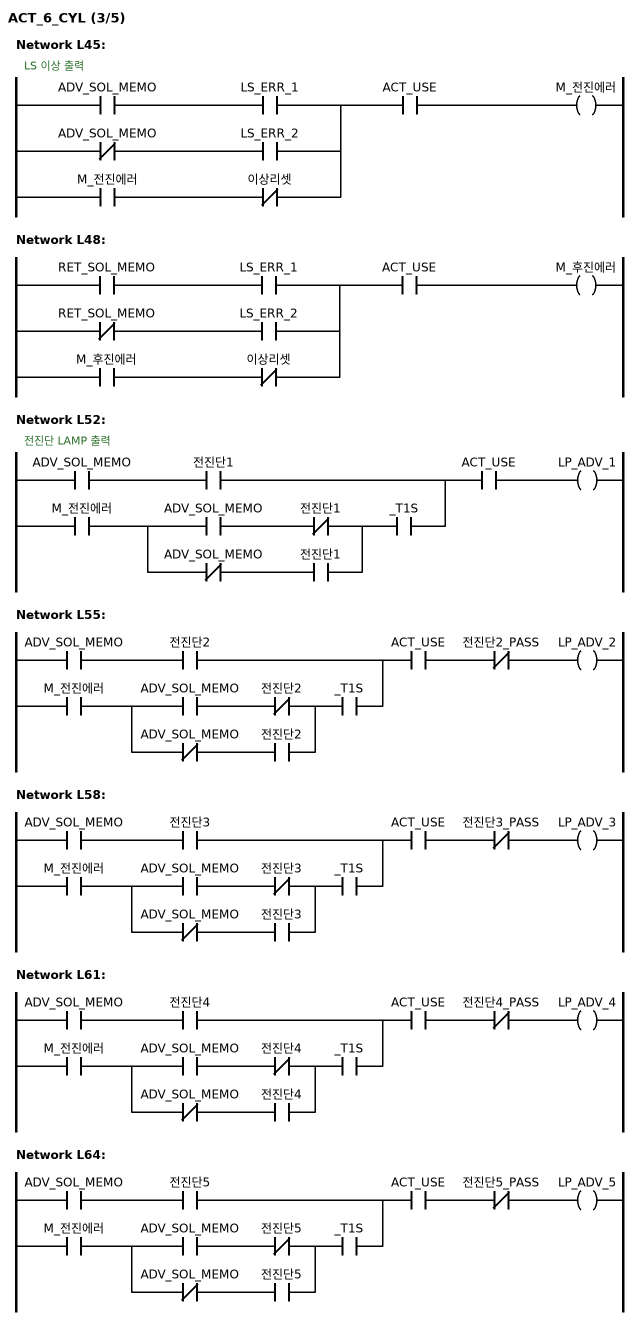
(* [picture p24: ACT_6_CYL rungs L45-L64] *)
(* LS 이상 출력 *)
(* Rung L45 *)
M_전진에러 := ((ADV_SOL_MEMO AND LS_ERR_1) OR (NOT ADV_SOL_MEMO AND LS_ERR_2) OR (M_전진에러 AND NOT 이상리셋)) AND ACT_USE;
(* Rung L48 *)
M_후진에러 := ((RET_SOL_MEMO AND LS_ERR_1) OR (NOT RET_SOL_MEMO AND LS_ERR_2) OR (M_후진에러 AND NOT 이상리셋)) AND ACT_USE;
(* 전진단 LAMP 출력 *)
(* Rung L52 *)
LP_ADV_1 := ((ADV_SOL_MEMO AND 전진단1) OR (M_전진에러 AND ((ADV_SOL_MEMO AND NOT 전진단1) OR (NOT ADV_SOL_MEMO AND 전진단1)) AND _T1S)) AND ACT_USE;
(* Rung L55 *)
LP_ADV_2 := ((ADV_SOL_MEMO AND 전진단2) OR (M_전진에러 AND ((ADV_SOL_MEMO AND NOT 전진단2) OR (NOT ADV_SOL_MEMO AND 전진단2)) AND _T1S)) AND ACT_USE AND NOT 전진단2_PASS;
(* Rung L58 *)
LP_ADV_3 := ((ADV_SOL_MEMO AND 전진단3) OR (M_전진에러 AND ((ADV_SOL_MEMO AND NOT 전진단3) OR (NOT ADV_SOL_MEMO AND 전진단3)) AND _T1S)) AND ACT_USE AND NOT 전진단3_PASS;
(* Rung L61 *)
LP_ADV_4 := ((ADV_SOL_MEMO AND 전진단4) OR (M_전진에러 AND ((ADV_SOL_MEMO AND NOT 전진단4) OR (NOT ADV_SOL_MEMO AND 전진단4)) AND _T1S)) AND ACT_USE AND NOT 전진단4_PASS;
(* Rung L64 *)
LP_ADV_5 := ((ADV_SOL_MEMO AND 전진단5) OR (M_전진에러 AND ((ADV_SOL_MEMO AND NOT 전진단5) OR (NOT ADV_SOL_MEMO AND 전진단5)) AND _T1S)) AND ACT_USE AND NOT 전진단5_PASS;

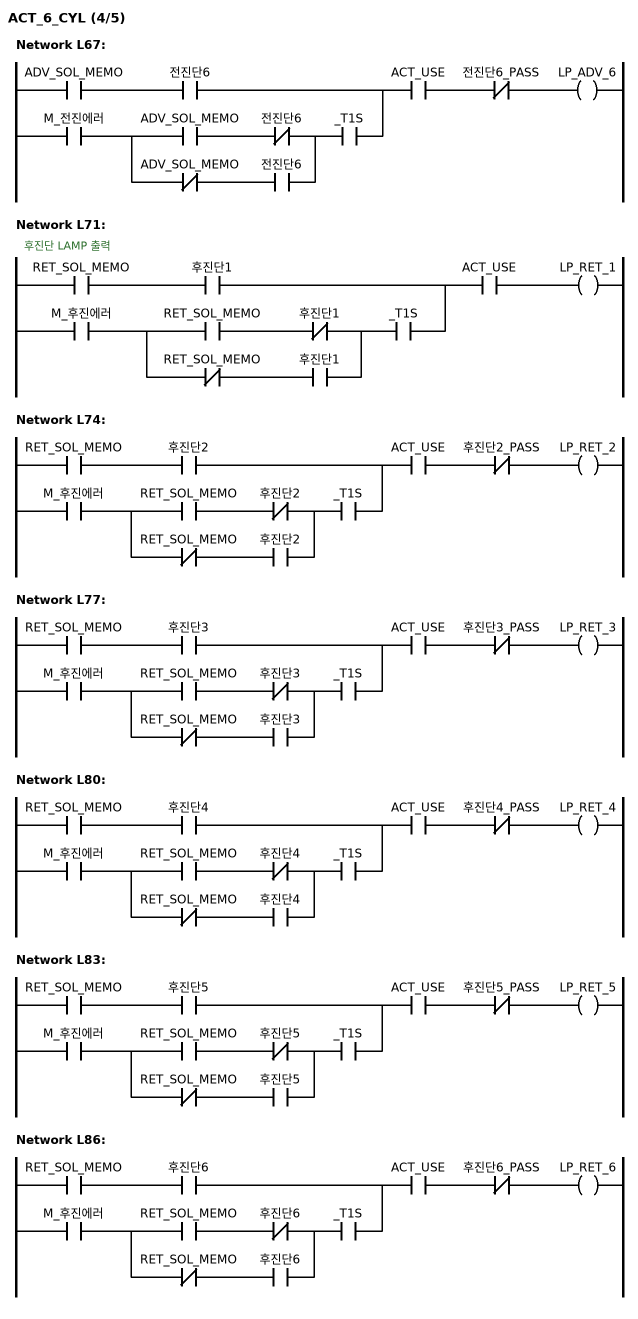
(* Rung L67 *)
LP_ADV_6 := ((ADV_SOL_MEMO AND 전진단6) OR (M_전진에러 AND ((ADV_SOL_MEMO AND NOT 전진단6) OR (NOT ADV_SOL_MEMO AND 전진단6)) AND _T1S)) AND ACT_USE AND NOT 전진단6_PASS;
(* 후진단 LAMP 출력 *)
(* Rung L71 *)
LP_RET_1 := ((RET_SOL_MEMO AND 후진단1) OR (M_후진에러 AND ((RET_SOL_MEMO AND NOT 후진단1) OR (NOT RET_SOL_MEMO AND 후진단1)) AND _T1S)) AND ACT_USE;
(* Rung L74 *)
LP_RET_2 := ((RET_SOL_MEMO AND 후진단2) OR (M_후진에러 AND ((RET_SOL_MEMO AND NOT 후진단2) OR (NOT RET_SOL_MEMO AND 후진단2)) AND _T1S)) AND ACT_USE AND NOT 후진단2_PASS;
(* Rung L77 *)
LP_RET_3 := ((RET_SOL_MEMO AND 후진단3) OR (M_후진에러 AND ((RET_SOL_MEMO AND NOT 후진단3) OR (NOT RET_SOL_MEMO AND 후진단3)) AND _T1S)) AND ACT_USE AND NOT 후진단3_PASS;
(* Rung L80 *)
LP_RET_4 := ((RET_SOL_MEMO AND 후진단4) OR (M_후진에러 AND ((RET_SOL_MEMO AND NOT 후진단4) OR (NOT RET_SOL_MEMO AND 후진단4)) AND _T1S)) AND ACT_USE AND NOT 후진단4_PASS;
(* Rung L83 *)
LP_RET_5 := ((RET_SOL_MEMO AND 후진단5) OR (M_후진에러 AND ((RET_SOL_MEMO AND NOT 후진단5) OR (NOT RET_SOL_MEMO AND 후진단5)) AND _T1S)) AND ACT_USE AND NOT 후진단5_PASS;
(* Rung L86 *)
LP_RET_6 := ((RET_SOL_MEMO AND 후진단6) OR (M_후진에러 AND ((RET_SOL_MEMO AND NOT 후진단6) OR (NOT RET_SOL_MEMO AND 후진단6)) AND _T1S)) AND ACT_USE AND NOT 후진단6_PASS;

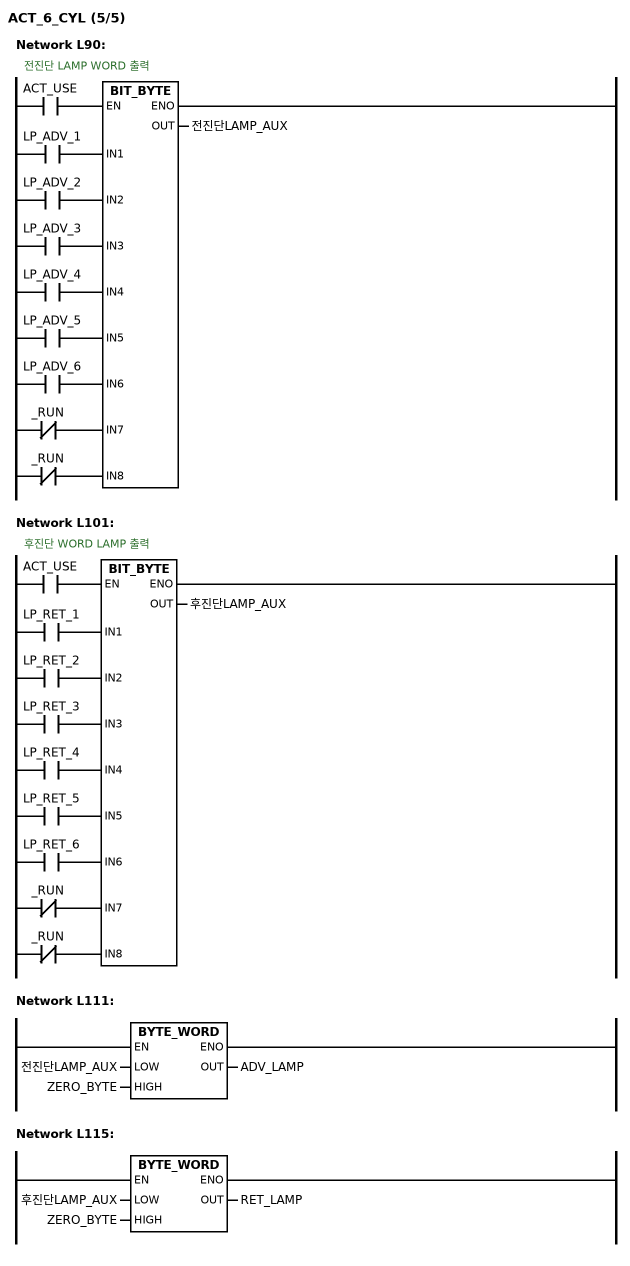
(* 전진단 LAMP WORD 출력 *)
(* Rung L90 *)
IF ACT_USE THEN
    전진단LAMP_AUX := BIT_BYTE(LP_ADV_1, LP_ADV_2, LP_ADV_3, LP_ADV_4, LP_ADV_5, LP_ADV_6, NOT _RUN, NOT _RUN);
END_IF;
(* 후진단 WORD LAMP 출력 *)
(* Rung L101 *)
IF ACT_USE THEN
    후진단LAMP_AUX := BIT_BYTE(LP_RET_1, LP_RET_2, LP_RET_3, LP_RET_4, LP_RET_5, LP_RET_6, NOT _RUN, NOT _RUN);
END_IF;
(* Rung L111 *)
ADV_LAMP := BYTE_WORD(LOW := 전진단LAMP_AUX, HIGH := ZERO_BYTE);
(* Rung L115 *)
RET_LAMP := BYTE_WORD(LOW := 후진단LAMP_AUX, HIGH := ZERO_BYTE);
END_FUNCTION_BLOCK

FUNCTION_BLOCK ACT_10_CYL
VAR_INPUT
    사용유무 : BOOL;
    운전준비 : BOOL;
    전진보조 : BOOL;
    후진보조 : BOOL;
    전진단수량 : UINT;
    후진단수량 : UINT;
    전진단1 : BOOL;
    후진단1 : BOOL;
    전진단2 : BOOL;
    후진단2 : BOOL;
    전진단3 : BOOL;
    후진단3 : BOOL;
    전진단4 : BOOL;
    후진단4 : BOOL;
    전진단5 : BOOL;
    후진단5 : BOOL;
    전진단6 : BOOL;
    후진단6 : BOOL;
    전진단7 : BOOL;
    후진단7 : BOOL;
    전진단8 : BOOL;
    후진단8 : BOOL;
    전진단9 : BOOL;
    후진단9 : BOOL;
    전진단10 : BOOL;
    후진단10 : BOOL;
    전진단_지연시간 : TIME;
    후진단_지연시간 : TIME;
    LS_ERR1_지연시간 : TIME;
    LS_ERR2_지연시간 : TIME;
    이상리셋 : BOOL;
END_VAR
VAR_OUTPUT
    SOL_ADV_출력 : BOOL;
    SOL_RET_출력 : BOOL;
    M_전진단 : BOOL;
    M_후진단 : BOOL;
    M_전진에러 : BOOL;
    M_후진에러 : BOOL;
    ADV_LAMP : WORD;
    RET_LAMP : WORD;
END_VAR
VAR
    ACT_USE : BOOL;
    ADV_END_TIME : TON;
    ADV_SOL_MEMO : BOOL;
    ERR_TIME1 : TON;
    LP_ADV_1 : BOOL;
    LP_ADV_10 : BOOL;
    LP_ADV_2 : BOOL;
    LP_ADV_3 : BOOL;
    LP_ADV_4 : BOOL;
    LP_ADV_5 : BOOL;
    LP_ADV_6 : BOOL;
    LP_ADV_7 : BOOL;
    LP_ADV_8 : BOOL;
    LP_ADV_9 : BOOL;
    LP_RET_1 : BOOL;
    LP_RET_10 : BOOL;
    LP_RET_2 : BOOL;
    LP_RET_3 : BOOL;
    LP_RET_4 : BOOL;
    LP_RET_5 : BOOL;
    LP_RET_6 : BOOL;
    LP_RET_7 : BOOL;
    LP_RET_8 : BOOL;
    LP_RET_9 : BOOL;
    LS_ERR_1 : BOOL;
    LS_ERR_2 : BOOL;
    RET_END_TIME : TON;
    RET_END_TIME1 : TON;
    RET_END_TIME2 : TON;
    RET_ERR_TIME : TON;
    RET_SOL_MEMO : BOOL;
    전진단10_PASS : BOOL;
    전진단2_PASS : BOOL;
    전진단3_PASS : BOOL;
    전진단4_PASS : BOOL;
    전진단5_PASS : BOOL;
    전진단6_PASS : BOOL;
    전진단7_PASS : BOOL;
    전진단8_PASS : BOOL;
    전진단9_PASS : BOOL;
    전진단LAMP_H_AUX : BYTE;
    전진단LAMP_L_AUX : BYTE;
    후진단10_PASS : BOOL;
    후진단2_PASS : BOOL;
    후진단3_PASS : BOOL;
    후진단4_PASS : BOOL;
    후진단5_PASS : BOOL;
    후진단6_PASS : BOOL;
    후진단7_PASS : BOOL;
    후진단8_PASS : BOOL;
    후진단9_PASS : BOOL;
    후진단LAMP_H_AUX : BYTE;
    후진단LAMP_L_AUX : BYTE;
END_VAR

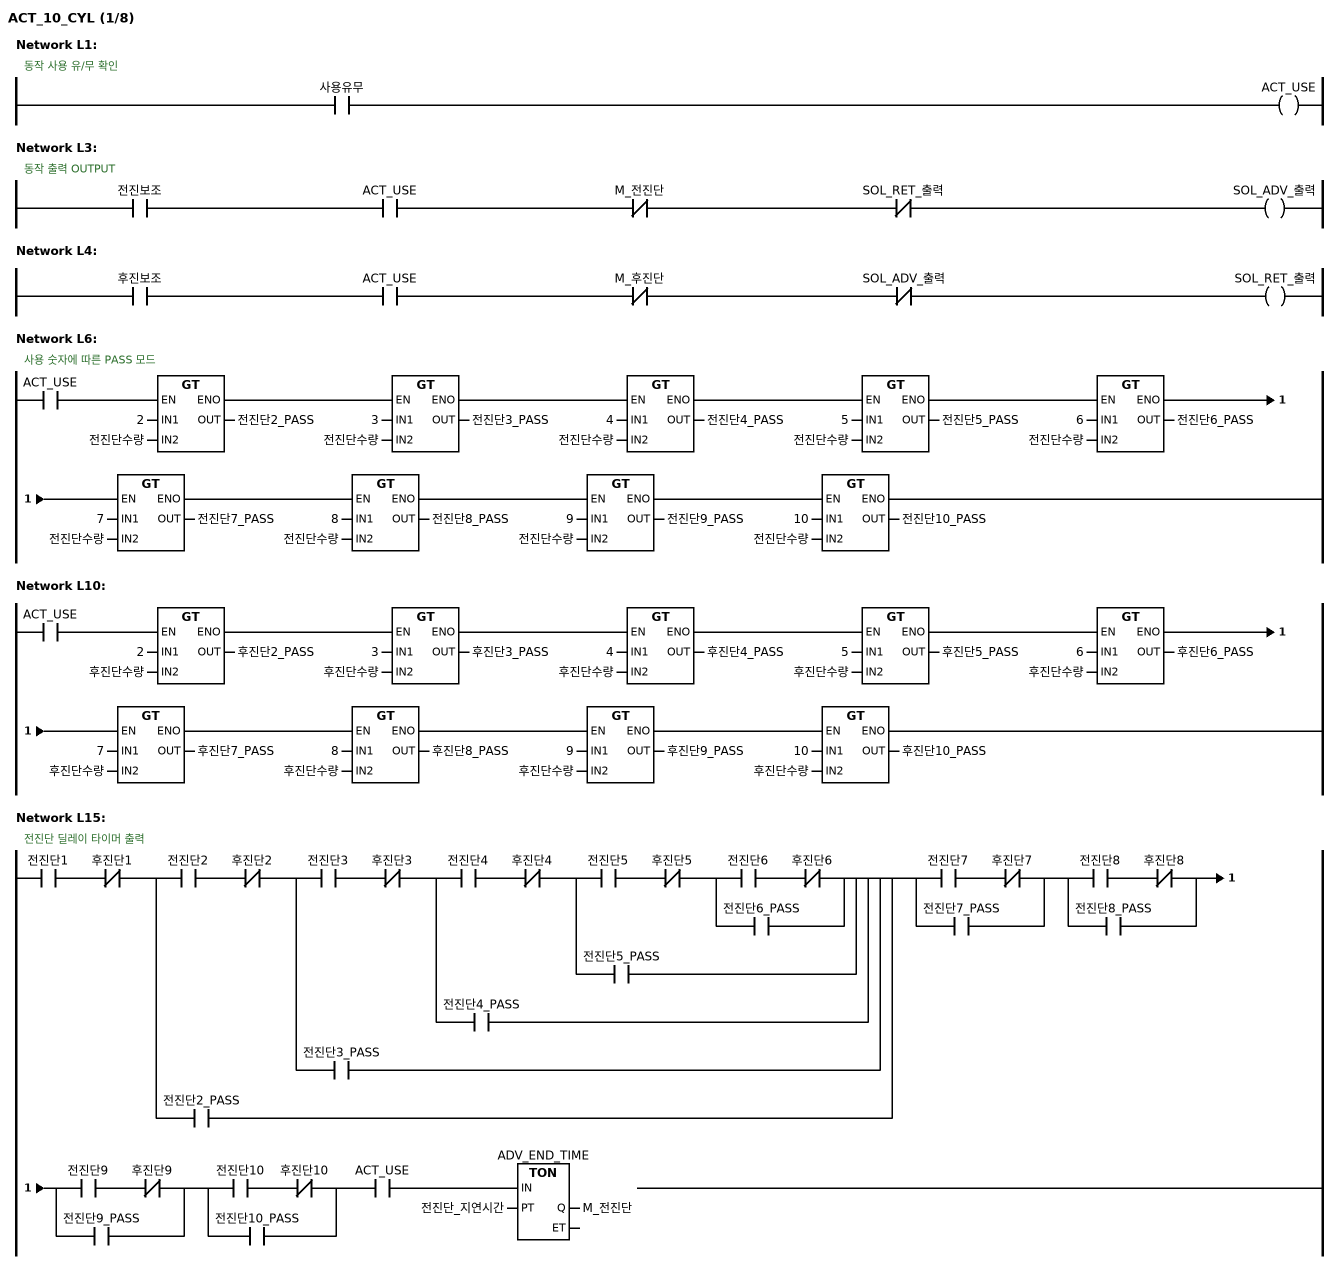
(* 동작 사용 유/무 확인 *)
(* Rung L1 *)
ACT_USE := 사용유무;
(* 동작 출력 OUTPUT *)
(* Rung L3 *)
SOL_ADV_출력 := 전진보조 AND ACT_USE AND NOT M_전진단 AND NOT SOL_RET_출력;
(* Rung L4 *)
SOL_RET_출력 := 후진보조 AND ACT_USE AND NOT M_후진단 AND NOT SOL_ADV_출력;
(* 사용 숫자에 따른 PASS 모드 *)
(* Rung L6 *)
IF ACT_USE THEN
    전진단2_PASS := 2 > 전진단수량;
    전진단3_PASS := 3 > 전진단수량;
    전진단4_PASS := 4 > 전진단수량;
    전진단5_PASS := 5 > 전진단수량;
    전진단6_PASS := 6 > 전진단수량;
    전진단7_PASS := 7 > 전진단수량;
    전진단8_PASS := 8 > 전진단수량;
    전진단9_PASS := 9 > 전진단수량;
    전진단10_PASS := 10 > 전진단수량;
END_IF;
(* Rung L10 *)
IF ACT_USE THEN
    후진단2_PASS := 2 > 후진단수량;
    후진단3_PASS := 3 > 후진단수량;
    후진단4_PASS := 4 > 후진단수량;
    후진단5_PASS := 5 > 후진단수량;
    후진단6_PASS := 6 > 후진단수량;
    후진단7_PASS := 7 > 후진단수량;
    후진단8_PASS := 8 > 후진단수량;
    후진단9_PASS := 9 > 후진단수량;
    후진단10_PASS := 10 > 후진단수량;
END_IF;
(* 전진단 딜레이 타이머 출력 *)
(* Rung L15 *)
ADV_END_TIME(IN := 전진단1 AND NOT 후진단1 AND ((전진단2 AND NOT 후진단2 AND ((전진단3 AND NOT 후진단3 AND ((전진단4 AND NOT 후진단4 AND ((전진단5 AND NOT 후진단5 AND ((전진단6 AND NOT 후진단6) OR 전진단6_PASS)) OR 전진단5_PASS)) OR 전진단4_PASS)) OR 전진단3_PASS)) OR 전진단2_PASS) AND ((전진단7 AND NOT 후진단7) OR 전진단7_PASS) AND ((전진단8 AND NOT 후진단8) OR 전진단8_PASS) AND ((전진단9 AND NOT 후진단9) OR 전진단9_PASS) AND ((전진단10 AND NOT 후진단10) OR 전진단10_PASS) AND ACT_USE, PT := 전진단_지연시간, Q => M_전진단);

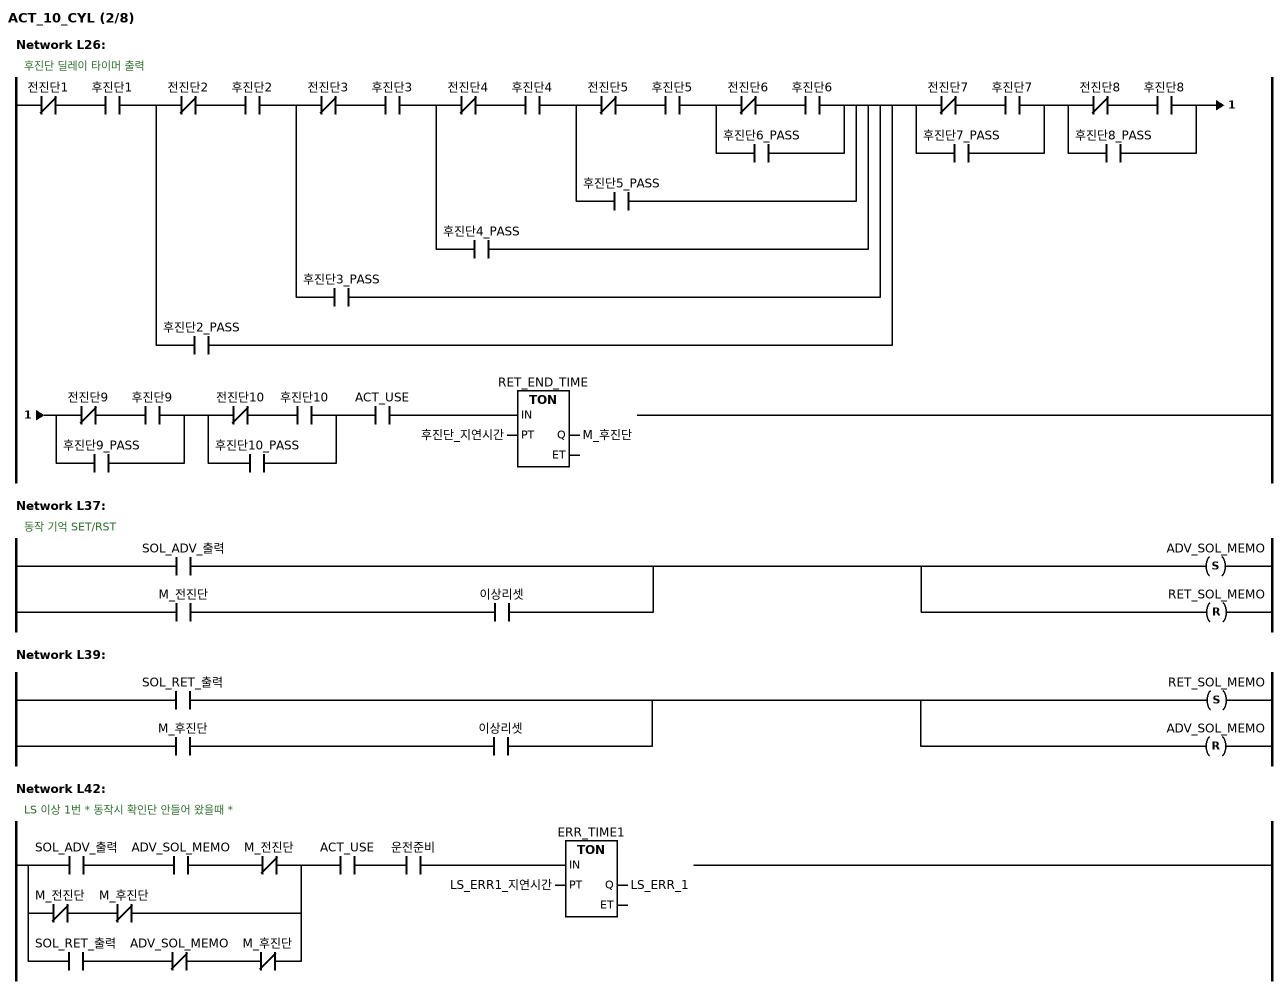
(* 후진단 딜레이 타이머 출력 *)
(* Rung L26 *)
RET_END_TIME(IN := NOT 전진단1 AND 후진단1 AND ((NOT 전진단2 AND 후진단2 AND ((NOT 전진단3 AND 후진단3 AND ((NOT 전진단4 AND 후진단4 AND ((NOT 전진단5 AND 후진단5 AND ((NOT 전진단6 AND 후진단6) OR 후진단6_PASS)) OR 후진단5_PASS)) OR 후진단4_PASS)) OR 후진단3_PASS)) OR 후진단2_PASS) AND ((NOT 전진단7 AND 후진단7) OR 후진단7_PASS) AND ((NOT 전진단8 AND 후진단8) OR 후진단8_PASS) AND ((NOT 전진단9 AND 후진단9) OR 후진단9_PASS) AND ((NOT 전진단10 AND 후진단10) OR 후진단10_PASS) AND ACT_USE, PT := 후진단_지연시간, Q => M_후진단);
(* 동작 기억 SET/RST *)
(* Rung L37 *)
IF SOL_ADV_출력 OR (M_전진단 AND 이상리셋) THEN
    ADV_SOL_MEMO := TRUE;
    RET_SOL_MEMO := FALSE;
END_IF;
(* Rung L39 *)
IF SOL_RET_출력 OR (M_후진단 AND 이상리셋) THEN
    RET_SOL_MEMO := TRUE;
    ADV_SOL_MEMO := FALSE;
END_IF;
(* LS 이상 1번 * 동작시 확인단 안들어 왔을때 * *)
(* Rung L42 *)
ERR_TIME1(IN := ((SOL_ADV_출력 AND ADV_SOL_MEMO AND NOT M_전진단) OR (NOT M_전진단 AND NOT M_후진단) OR (SOL_RET_출력 AND NOT ADV_SOL_MEMO AND NOT M_후진단)) AND ACT_USE AND 운전준비, PT := LS_ERR1_지연시간, Q => LS_ERR_1);

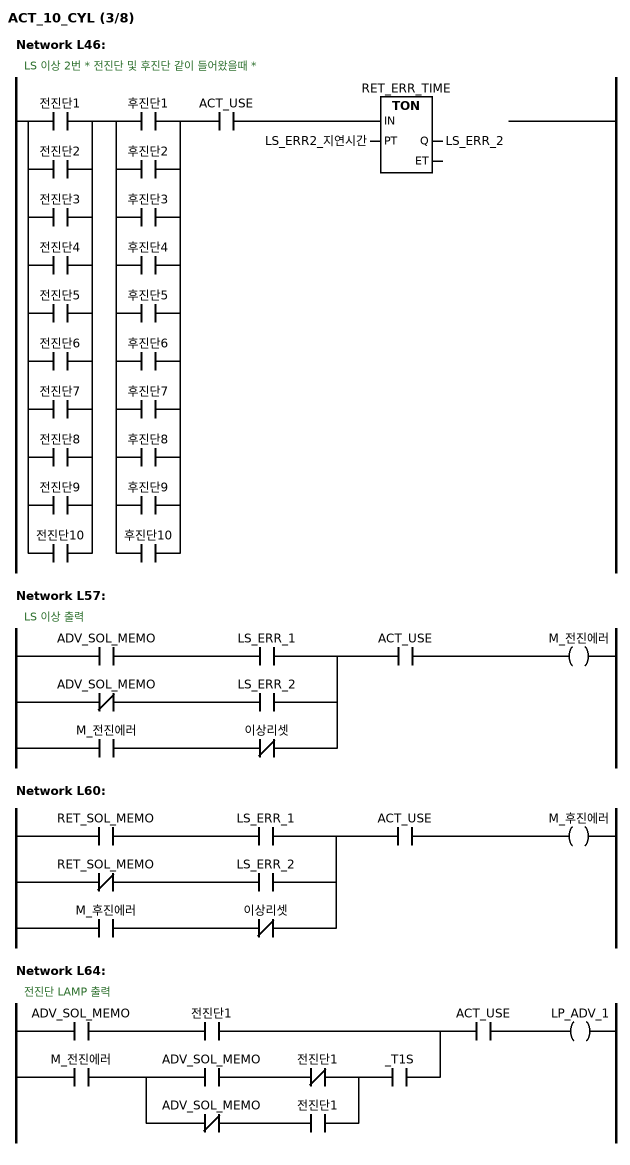
(* LS 이상 2번 * 전진단 및 후진단 같이 들어왔을때 * *)
(* Rung L46 *)
RET_ERR_TIME(IN := (전진단1 OR 전진단2 OR 전진단3 OR 전진단4 OR 전진단5 OR 전진단6 OR 전진단7 OR 전진단8 OR 전진단9 OR 전진단10) AND (후진단1 OR 후진단2 OR 후진단3 OR 후진단4 OR 후진단5 OR 후진단6 OR 후진단7 OR 후진단8 OR 후진단9 OR 후진단10) AND ACT_USE, PT := LS_ERR2_지연시간, Q => LS_ERR_2);
(* LS 이상 출력 *)
(* Rung L57 *)
M_전진에러 := ((ADV_SOL_MEMO AND LS_ERR_1) OR (NOT ADV_SOL_MEMO AND LS_ERR_2) OR (M_전진에러 AND NOT 이상리셋)) AND ACT_USE;
(* Rung L60 *)
M_후진에러 := ((RET_SOL_MEMO AND LS_ERR_1) OR (NOT RET_SOL_MEMO AND LS_ERR_2) OR (M_후진에러 AND NOT 이상리셋)) AND ACT_USE;
(* 전진단 LAMP 출력 *)
(* Rung L64 *)
LP_ADV_1 := ((ADV_SOL_MEMO AND 전진단1) OR (M_전진에러 AND ((ADV_SOL_MEMO AND NOT 전진단1) OR (NOT ADV_SOL_MEMO AND 전진단1)) AND _T1S)) AND ACT_USE;

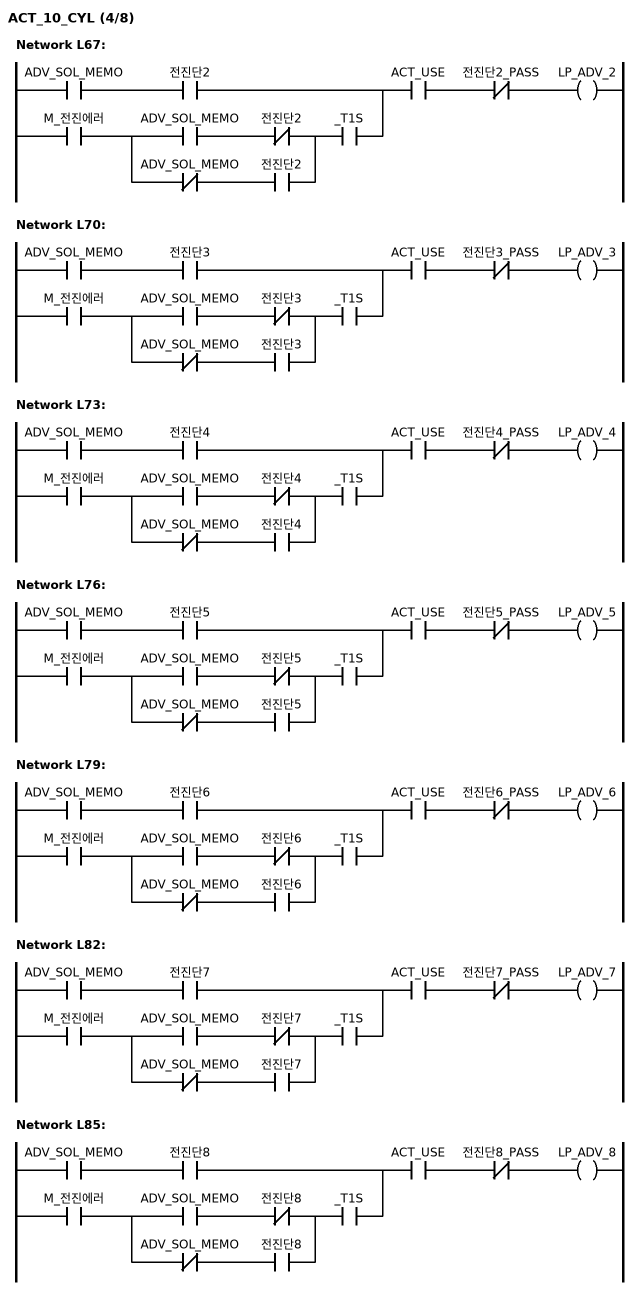
(* Rung L67 *)
LP_ADV_2 := ((ADV_SOL_MEMO AND 전진단2) OR (M_전진에러 AND ((ADV_SOL_MEMO AND NOT 전진단2) OR (NOT ADV_SOL_MEMO AND 전진단2)) AND _T1S)) AND ACT_USE AND NOT 전진단2_PASS;
(* Rung L70 *)
LP_ADV_3 := ((ADV_SOL_MEMO AND 전진단3) OR (M_전진에러 AND ((ADV_SOL_MEMO AND NOT 전진단3) OR (NOT ADV_SOL_MEMO AND 전진단3)) AND _T1S)) AND ACT_USE AND NOT 전진단3_PASS;
(* Rung L73 *)
LP_ADV_4 := ((ADV_SOL_MEMO AND 전진단4) OR (M_전진에러 AND ((ADV_SOL_MEMO AND NOT 전진단4) OR (NOT ADV_SOL_MEMO AND 전진단4)) AND _T1S)) AND ACT_USE AND NOT 전진단4_PASS;
(* Rung L76 *)
LP_ADV_5 := ((ADV_SOL_MEMO AND 전진단5) OR (M_전진에러 AND ((ADV_SOL_MEMO AND NOT 전진단5) OR (NOT ADV_SOL_MEMO AND 전진단5)) AND _T1S)) AND ACT_USE AND NOT 전진단5_PASS;
(* Rung L79 *)
LP_ADV_6 := ((ADV_SOL_MEMO AND 전진단6) OR (M_전진에러 AND ((ADV_SOL_MEMO AND NOT 전진단6) OR (NOT ADV_SOL_MEMO AND 전진단6)) AND _T1S)) AND ACT_USE AND NOT 전진단6_PASS;
(* Rung L82 *)
LP_ADV_7 := ((ADV_SOL_MEMO AND 전진단7) OR (M_전진에러 AND ((ADV_SOL_MEMO AND NOT 전진단7) OR (NOT ADV_SOL_MEMO AND 전진단7)) AND _T1S)) AND ACT_USE AND NOT 전진단7_PASS;
(* Rung L85 *)
LP_ADV_8 := ((ADV_SOL_MEMO AND 전진단8) OR (M_전진에러 AND ((ADV_SOL_MEMO AND NOT 전진단8) OR (NOT ADV_SOL_MEMO AND 전진단8)) AND _T1S)) AND ACT_USE AND NOT 전진단8_PASS;

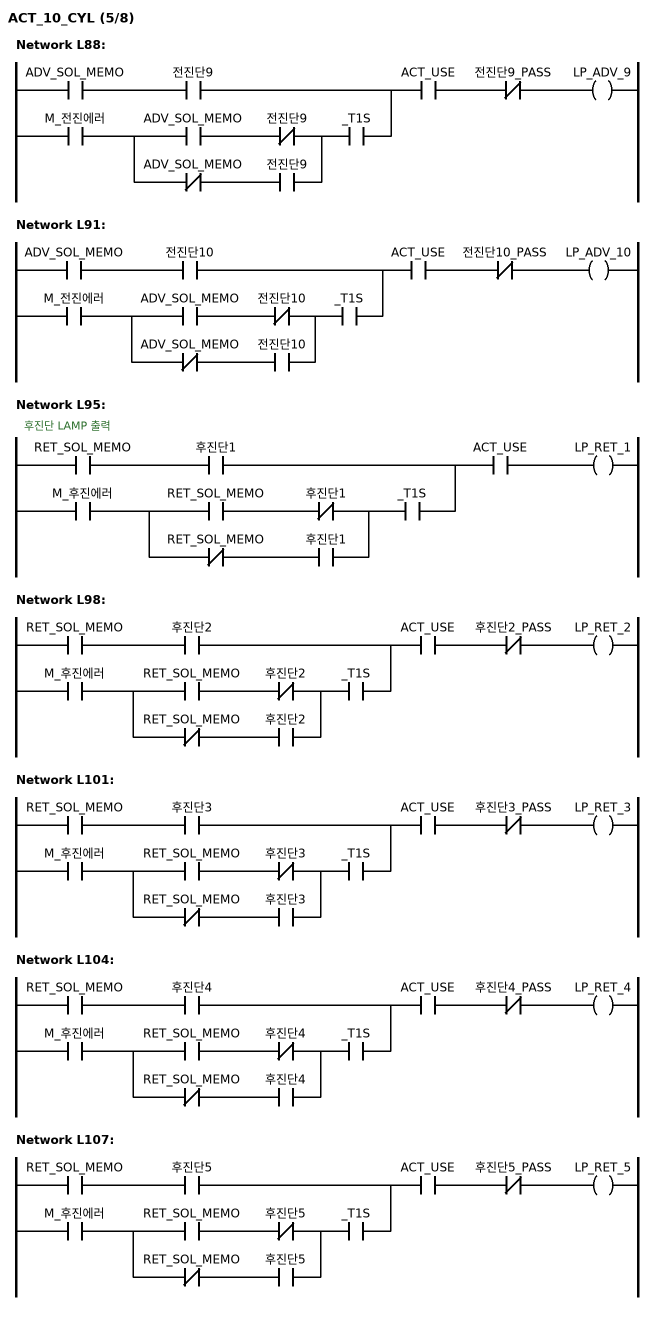
(* Rung L88 *)
LP_ADV_9 := ((ADV_SOL_MEMO AND 전진단9) OR (M_전진에러 AND ((ADV_SOL_MEMO AND NOT 전진단9) OR (NOT ADV_SOL_MEMO AND 전진단9)) AND _T1S)) AND ACT_USE AND NOT 전진단9_PASS;
(* Rung L91 *)
LP_ADV_10 := ((ADV_SOL_MEMO AND 전진단10) OR (M_전진에러 AND ((ADV_SOL_MEMO AND NOT 전진단10) OR (NOT ADV_SOL_MEMO AND 전진단10)) AND _T1S)) AND ACT_USE AND NOT 전진단10_PASS;
(* 후진단 LAMP 출력 *)
(* Rung L95 *)
LP_RET_1 := ((RET_SOL_MEMO AND 후진단1) OR (M_후진에러 AND ((RET_SOL_MEMO AND NOT 후진단1) OR (NOT RET_SOL_MEMO AND 후진단1)) AND _T1S)) AND ACT_USE;
(* Rung L98 *)
LP_RET_2 := ((RET_SOL_MEMO AND 후진단2) OR (M_후진에러 AND ((RET_SOL_MEMO AND NOT 후진단2) OR (NOT RET_SOL_MEMO AND 후진단2)) AND _T1S)) AND ACT_USE AND NOT 후진단2_PASS;
(* Rung L101 *)
LP_RET_3 := ((RET_SOL_MEMO AND 후진단3) OR (M_후진에러 AND ((RET_SOL_MEMO AND NOT 후진단3) OR (NOT RET_SOL_MEMO AND 후진단3)) AND _T1S)) AND ACT_USE AND NOT 후진단3_PASS;
(* Rung L104 *)
LP_RET_4 := ((RET_SOL_MEMO AND 후진단4) OR (M_후진에러 AND ((RET_SOL_MEMO AND NOT 후진단4) OR (NOT RET_SOL_MEMO AND 후진단4)) AND _T1S)) AND ACT_USE AND NOT 후진단4_PASS;
(* Rung L107 *)
LP_RET_5 := ((RET_SOL_MEMO AND 후진단5) OR (M_후진에러 AND ((RET_SOL_MEMO AND NOT 후진단5) OR (NOT RET_SOL_MEMO AND 후진단5)) AND _T1S)) AND ACT_USE AND NOT 후진단5_PASS;

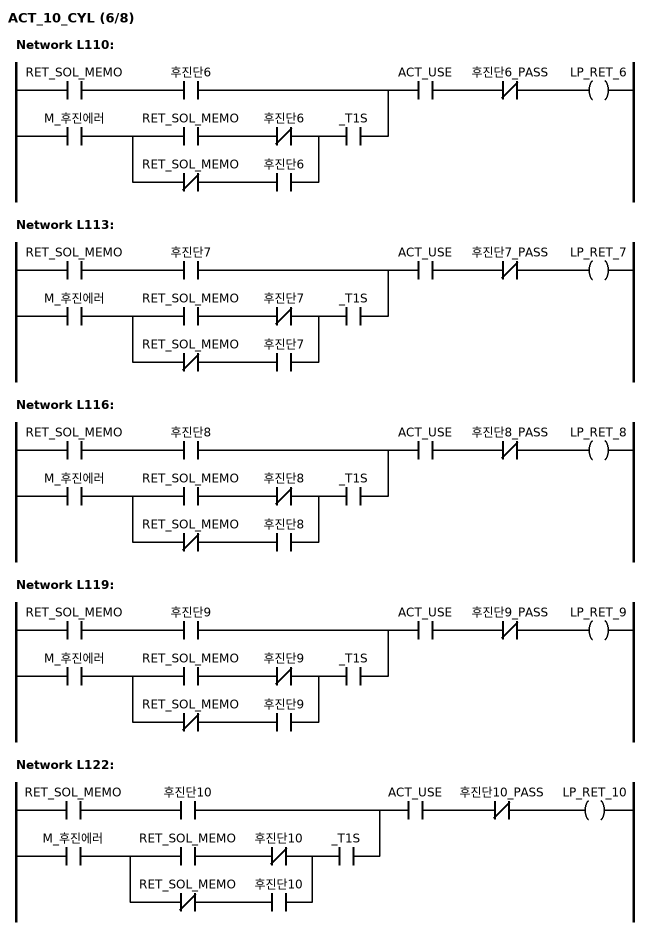
(* Rung L110 *)
LP_RET_6 := ((RET_SOL_MEMO AND 후진단6) OR (M_후진에러 AND ((RET_SOL_MEMO AND NOT 후진단6) OR (NOT RET_SOL_MEMO AND 후진단6)) AND _T1S)) AND ACT_USE AND NOT 후진단6_PASS;
(* Rung L113 *)
LP_RET_7 := ((RET_SOL_MEMO AND 후진단7) OR (M_후진에러 AND ((RET_SOL_MEMO AND NOT 후진단7) OR (NOT RET_SOL_MEMO AND 후진단7)) AND _T1S)) AND ACT_USE AND NOT 후진단7_PASS;
(* Rung L116 *)
LP_RET_8 := ((RET_SOL_MEMO AND 후진단8) OR (M_후진에러 AND ((RET_SOL_MEMO AND NOT 후진단8) OR (NOT RET_SOL_MEMO AND 후진단8)) AND _T1S)) AND ACT_USE AND NOT 후진단8_PASS;
(* Rung L119 *)
LP_RET_9 := ((RET_SOL_MEMO AND 후진단9) OR (M_후진에러 AND ((RET_SOL_MEMO AND NOT 후진단9) OR (NOT RET_SOL_MEMO AND 후진단9)) AND _T1S)) AND ACT_USE AND NOT 후진단9_PASS;
(* Rung L122 *)
LP_RET_10 := ((RET_SOL_MEMO AND 후진단10) OR (M_후진에러 AND ((RET_SOL_MEMO AND NOT 후진단10) OR (NOT RET_SOL_MEMO AND 후진단10)) AND _T1S)) AND ACT_USE AND NOT 후진단10_PASS;

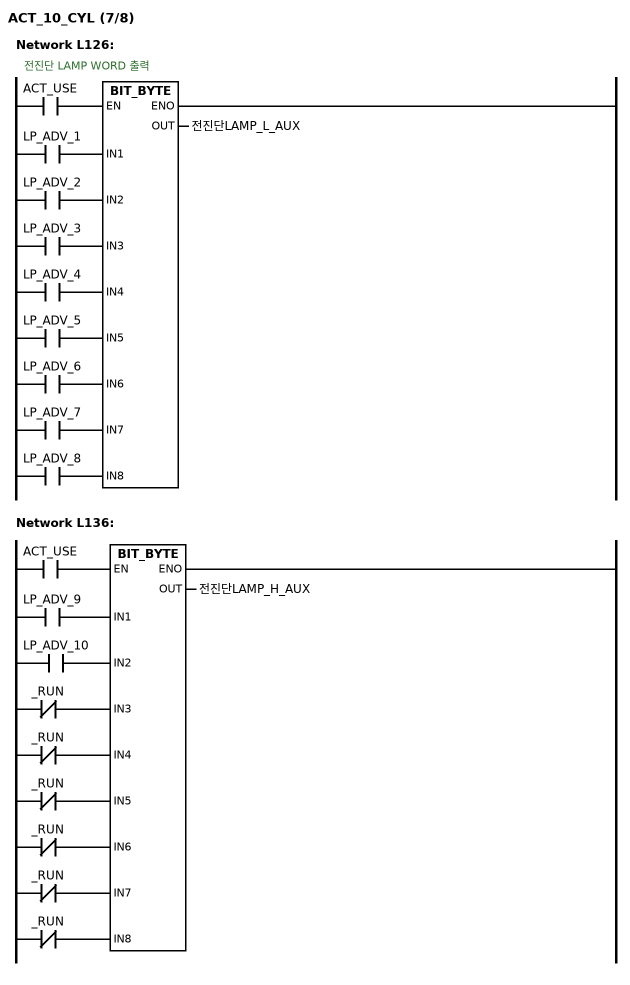
(* 전진단 LAMP WORD 출력 *)
(* Rung L126 *)
IF ACT_USE THEN
    전진단LAMP_L_AUX := BIT_BYTE(LP_ADV_1, LP_ADV_2, LP_ADV_3, LP_ADV_4, LP_ADV_5, LP_ADV_6, LP_ADV_7, LP_ADV_8);
END_IF;
(* Rung L136 *)
IF ACT_USE THEN
    전진단LAMP_H_AUX := BIT_BYTE(LP_ADV_9, LP_ADV_10, NOT _RUN, NOT _RUN, NOT _RUN, NOT _RUN, NOT _RUN, NOT _RUN);
END_IF;

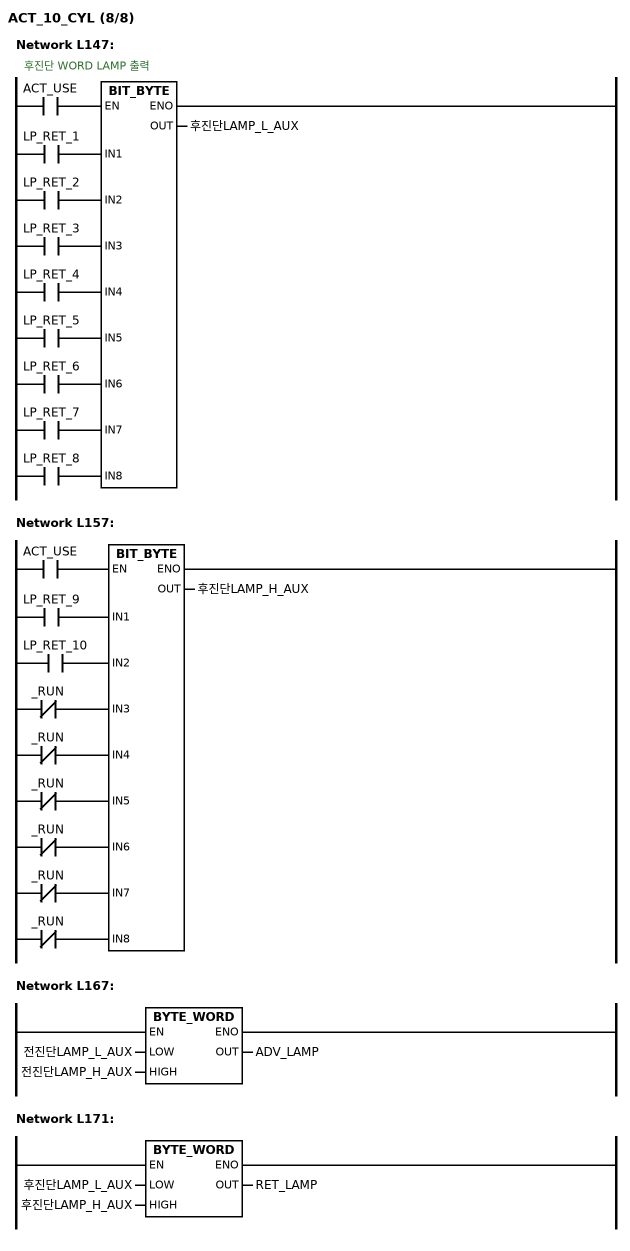
(* 후진단 WORD LAMP 출력 *)
(* Rung L147 *)
IF ACT_USE THEN
    후진단LAMP_L_AUX := BIT_BYTE(LP_RET_1, LP_RET_2, LP_RET_3, LP_RET_4, LP_RET_5, LP_RET_6, LP_RET_7, LP_RET_8);
END_IF;
(* Rung L157 *)
IF ACT_USE THEN
    후진단LAMP_H_AUX := BIT_BYTE(LP_RET_9, LP_RET_10, NOT _RUN, NOT _RUN, NOT _RUN, NOT _RUN, NOT _RUN, NOT _RUN);
END_IF;
(* Rung L167 *)
ADV_LAMP := BYTE_WORD(LOW := 전진단LAMP_L_AUX, HIGH := 전진단LAMP_H_AUX);
(* Rung L171 *)
RET_LAMP := BYTE_WORD(LOW := 후진단LAMP_L_AUX, HIGH := 후진단LAMP_H_AUX);
END_FUNCTION_BLOCK

PROGRAM 운전모드 (* task: 스캔 프로그램 *)
VAR_EXTERNAL
    AWAYS_ON : BOOL; (* AT %MW3.1 *)
    CLOCK_BIT_0_5Sec : BOOL; (* AT %MW0.3 *)
    EGIS_EJS : BOOL;
    GATE10_M_도어_잠김 : BOOL; (* AT %MW409.3 *)
    GATE10_M_비상정지 : BOOL; (* AT %MW409.7 *)
    GATE10_M_이상_리셋 : BOOL; (* AT %MW409.0 *)
    GATE10_M_정상 : BOOL; (* AT %MW409.4 *)
    GATE11_M_이상_리셋 : BOOL; (* AT %MW410.0 *)
    GATE11_M_정상 : BOOL; (* AT %MW410.4 *)
    GATE12_M_이상_리셋 : BOOL; (* AT %MW411.0 *)
    GATE12_M_정상 : BOOL; (* AT %MW411.4 *)
    MCP_EPB_비상정지1 : BOOL; (* AT %MW87635.0 *) (* 입력 접점 00 *)
    MCP_EPB_비상정지2 : BOOL; (* AT %MW87635.1 *) (* 입력 접점 01 *)
    MCP_KSW_MES_OFF : BOOL; (* AT %MW87631.4 *) (* 입력 접점 04 *)
    MCP_KSW_MES_ON : BOOL; (* AT %MW87631.5 *) (* 입력 접점 05 *)
    MCP_MC1_OUTPUT_PWR_ON : BOOL; (* AT %MW97636.0 *) (* 출력 접점 00 *)
    MCP_M_램프_테스트 : BOOL; (* AT %MW350.6 *)
    MCP_M_부저_정지 : BOOL; (* AT %MW350.5 *)
    MCP_M_비상정지 : BOOL; (* AT %MW350.7 *)
    MCP_M_수동_모드 : BOOL; (* AT %MW350.1 *)
    MCP_M_운전준비_ON : BOOL; (* AT %MW350.0 *)
    MCP_M_이상_리셋 : BOOL; (* AT %MW350.4 *)
    MCP_M_자동_START : BOOL; (* AT %MW350.3 *)
    MCP_M_자동_모드 : BOOL; (* AT %MW350.2 *)
    MCP_PBL_101_자동_운전 : BOOL; (* AT %MW87630.4 *) (* 입력 접점 04 *)
    MCP_PBL_101_자동_운전_LP : BOOL; (* AT %MW97633.1 *) (* 출력 접점 01 *)
    MCP_PBL_102_자동_운전 : BOOL; (* AT %MW87630.7 *) (* 입력 접점 07 *)
    MCP_PBL_102_자동_운전_LP : BOOL; (* AT %MW97633.2 *) (* 출력 접점 02 *)
    MCP_PBL_103_4_자동_운전 : BOOL; (* AT %MW87630.10 *) (* 입력 접점 10 *)
    MCP_PBL_103_4_자동_운전_LP : BOOL; (* AT %MW97633.3 *) (* 출력 접점 03 *)
    MCP_PBL_운전준비_ON : BOOL; (* AT %MW87630.0 *) (* 입력 접점 00 *)
    MCP_PBL_운전준비_ON_LP : BOOL; (* AT %MW97633.0 *) (* 출력 접점 00 *)
    MCP_PB_이상_리셋 : BOOL; (* AT %MW87630.1 *) (* 입력 접점 01 *)
    MCP_SPB_램프_테스트 : BOOL; (* AT %MW87631.2 *) (* 입력 접점 02 *)
    MCP_SPB_부저_정지 : BOOL; (* AT %MW87631.3 *) (* 입력 접점 03 *)
    MCP_SPK_MEL1 : BOOL; (* AT %MW97633.8 *) (* 출력 접점 08 *)
    MCP_SSP_101_수동_선택 : BOOL; (* AT %MW87630.2 *) (* 입력 접점 02 *)
    MCP_SSP_101_자동_선택 : BOOL; (* AT %MW87630.3 *) (* 입력 접점 03 *)
    MCP_TL_GREEN_LAMP : BOOL; (* AT %MW97633.6 *) (* 출력 접점 06 *)
    MCP_TL_RED_LAMP : BOOL; (* AT %MW97633.4 *) (* 출력 접점 04 *)
    MCP_TL_YELLOW_LAMP : BOOL; (* AT %MW97633.5 *) (* 출력 접점 05 *)
    MCP_타워_부저 : BOOL; (* AT %MW97633.7 *) (* 출력 접점 07 *)
    S101_M_수동_모드 : BOOL; (* AT %MW1000.3 *)
    S101_M_운전준비_ON : BOOL; (* AT %MW1000.0 *)
    S101_M_자동_START : BOOL; (* AT %MW1000.5 *)
    S101_M_자동_모드 : BOOL; (* AT %MW1000.1 *)
    S101_M_자동_운전중 : BOOL; (* AT %MW1000.4 *)
    S101_M_총괄_비상정지_이상 : BOOL; (* AT %MW1009.1 *)
    S101_M_총괄_이상 : BOOL; (* AT %MW1009.0 *)
    S102_M_수동_모드 : BOOL; (* AT %MW1500.3 *)
    S102_M_운전준비_ON : BOOL; (* AT %MW1500.0 *)
    S102_M_자동_START : BOOL; (* AT %MW1500.5 *)
    S102_M_자동_모드 : BOOL; (* AT %MW1500.1 *)
    S102_M_자동_운전중 : BOOL; (* AT %MW1500.4 *)
    S102_M_총괄_비상정지_이상 : BOOL; (* AT %MW1509.1 *)
    S102_M_총괄_이상 : BOOL; (* AT %MW1509.0 *)
    S103_M_수동_모드 : BOOL; (* AT %MW2000.3 *)
    S103_M_운전준비_ON : BOOL; (* AT %MW2000.0 *)
    S103_M_자동_START : BOOL; (* AT %MW2000.5 *)
    S103_M_자동_모드 : BOOL; (* AT %MW2000.1 *)
    S103_M_자동_운전중 : BOOL; (* AT %MW2000.4 *)
    S103_M_총괄_비상정지_이상 : BOOL; (* AT %MW2009.1 *)
    S103_M_총괄_이상 : BOOL; (* AT %MW2009.0 *)
    S104_M_수동_모드 : BOOL; (* AT %MW2500.3 *)
    S104_M_운전준비_ON : BOOL; (* AT %MW2500.0 *)
    S104_M_자동_START : BOOL; (* AT %MW2500.5 *)
    S104_M_자동_모드 : BOOL; (* AT %MW2500.1 *)
    S104_M_총괄_비상정지_이상 : BOOL; (* AT %MW2509.1 *)
    S104_M_총괄_이상 : BOOL; (* AT %MW2509.0 *)
    T101_자동 : TON;
    T102_자동 : TON;
    TON_부저_정지 : TON;
    TON_부저_정지1 : TON;
    전체_M_운전준비_보조 : BOOL; (* AT %MW308.5 *)
    전체_M_이상_리셋 : BOOL; (* AT %MW308.2 *) (* 전체 M 이상 리셋 *)
    전체_라인_M_총괄_ROBOT_이상 : BOOL; (* AT %MW301.1 *)
    전체_라인_M_총괄_SAFETY_이상 : BOOL; (* AT %MW300.2 *)
    전체_라인_M_총괄_공기압_이상 : BOOL; (* AT %MW300.3 *)
    전체_라인_M_총괄_비상정지_이상 : BOOL; (* AT %MW300.1 *)
    전체_라인_M_총괄_이상 : BOOL; (* AT %MW300.0 *)
END_VAR
VAR
    시운전모드 : BOOL;
END_VAR
VAR
    _p1 : BOOL;
END_VAR

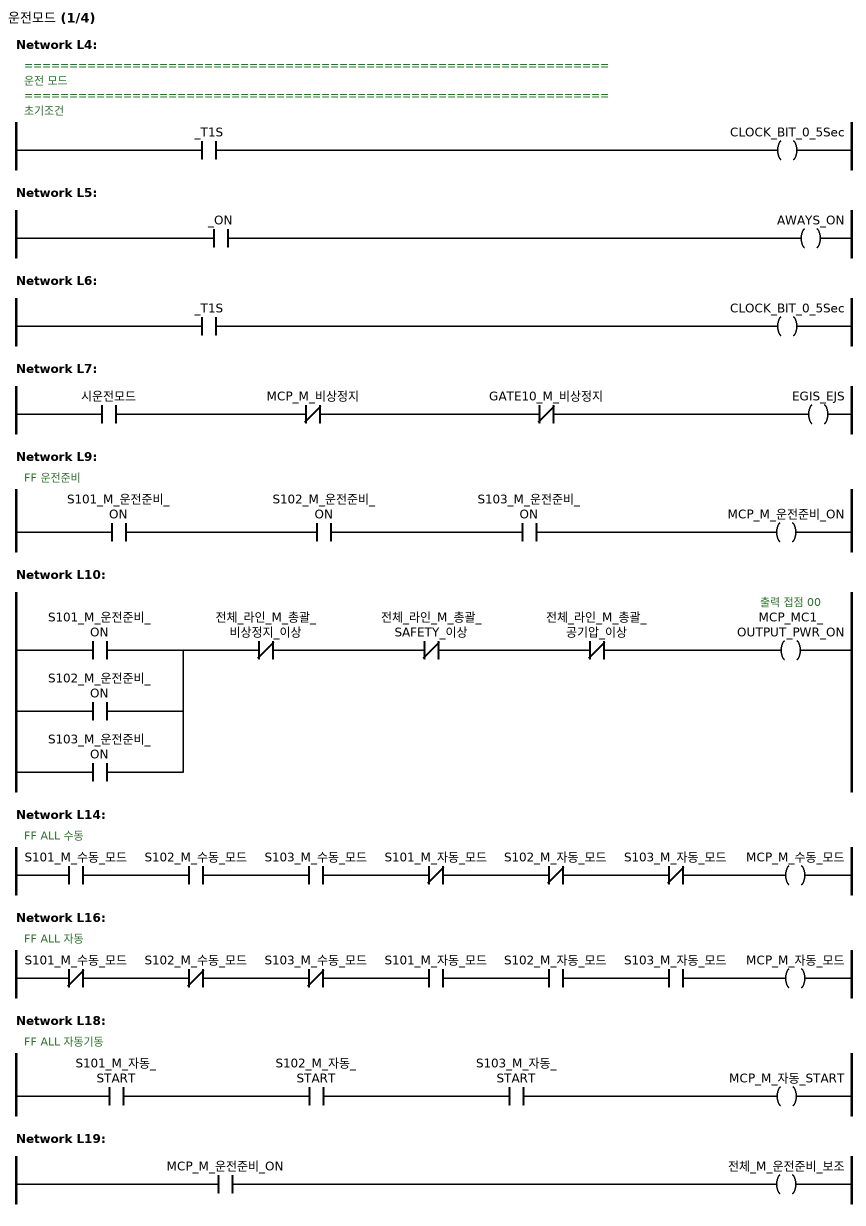
(* ================================================================= *)
(* 운전 모드 *)
(* ================================================================= *)
(* 초기조건 *)
(* Rung L4 *)
CLOCK_BIT_0_5Sec := _T1S;
(* Rung L5 *)
AWAYS_ON := _ON;
(* Rung L6 *)
CLOCK_BIT_0_5Sec := _T1S;
(* Rung L7 *)
EGIS_EJS := 시운전모드 AND NOT MCP_M_비상정지 AND NOT GATE10_M_비상정지;
(* FF 운전준비 *)
(* Rung L9 *)
MCP_M_운전준비_ON := S101_M_운전준비_ON AND S102_M_운전준비_ON AND S103_M_운전준비_ON;
(* Rung L10 *)
MCP_MC1_OUTPUT_PWR_ON := (S101_M_운전준비_ON OR S102_M_운전준비_ON OR S103_M_운전준비_ON) AND NOT 전체_라인_M_총괄_비상정지_이상 AND NOT 전체_라인_M_총괄_SAFETY_이상 AND NOT 전체_라인_M_총괄_공기압_이상;
(* FF ALL 수동 *)
(* Rung L14 *)
MCP_M_수동_모드 := S101_M_수동_모드 AND S102_M_수동_모드 AND S103_M_수동_모드 AND NOT S101_M_자동_모드 AND NOT S102_M_자동_모드 AND NOT S103_M_자동_모드;
(* FF ALL 자동 *)
(* Rung L16 *)
MCP_M_자동_모드 := NOT S101_M_수동_모드 AND NOT S102_M_수동_모드 AND NOT S103_M_수동_모드 AND S101_M_자동_모드 AND S102_M_자동_모드 AND S103_M_자동_모드;
(* FF ALL 자동기동 *)
(* Rung L18 *)
MCP_M_자동_START := S101_M_자동_START AND S102_M_자동_START AND S103_M_자동_START;
(* Rung L19 *)
전체_M_운전준비_보조 := MCP_M_운전준비_ON;

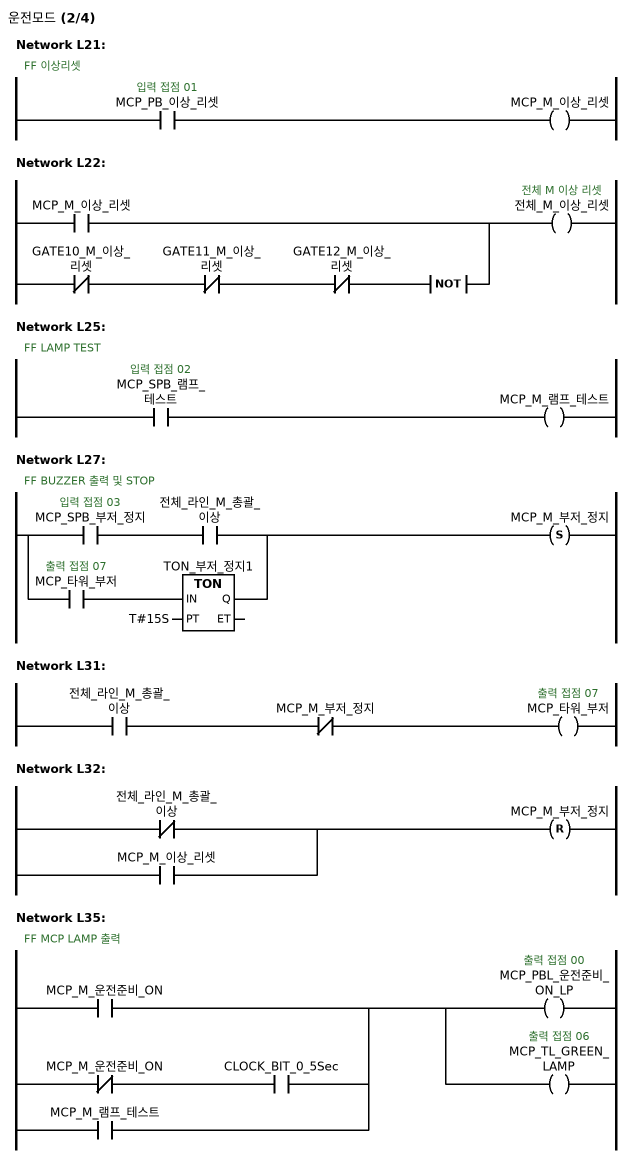
(* FF 이상리셋 *)
(* Rung L21 *)
MCP_M_이상_리셋 := MCP_PB_이상_리셋;
(* Rung L22 *)
전체_M_이상_리셋 := MCP_M_이상_리셋 OR NOT (NOT GATE10_M_이상_리셋 AND NOT GATE11_M_이상_리셋 AND NOT GATE12_M_이상_리셋);
(* FF LAMP TEST *)
(* Rung L25 *)
MCP_M_램프_테스트 := MCP_SPB_램프_테스트;
(* FF BUZZER 출력 및 STOP *)
(* Rung L27 *)
TON_부저_정지1(IN := MCP_타워_부저, PT := T#15S);
IF (MCP_SPB_부저_정지 AND 전체_라인_M_총괄_이상) OR TON_부저_정지1.Q THEN MCP_M_부저_정지 := TRUE; END_IF;
(* Rung L31 *)
MCP_타워_부저 := 전체_라인_M_총괄_이상 AND NOT MCP_M_부저_정지;
(* Rung L32 *)
IF NOT 전체_라인_M_총괄_이상 OR MCP_M_이상_리셋 THEN MCP_M_부저_정지 := FALSE; END_IF;
(* FF MCP LAMP 출력 *)
(* Rung L35 *)
_p1 := MCP_M_운전준비_ON OR (NOT MCP_M_운전준비_ON AND CLOCK_BIT_0_5Sec) OR MCP_M_램프_테스트;
MCP_PBL_운전준비_ON_LP := _p1;
MCP_TL_GREEN_LAMP := _p1;

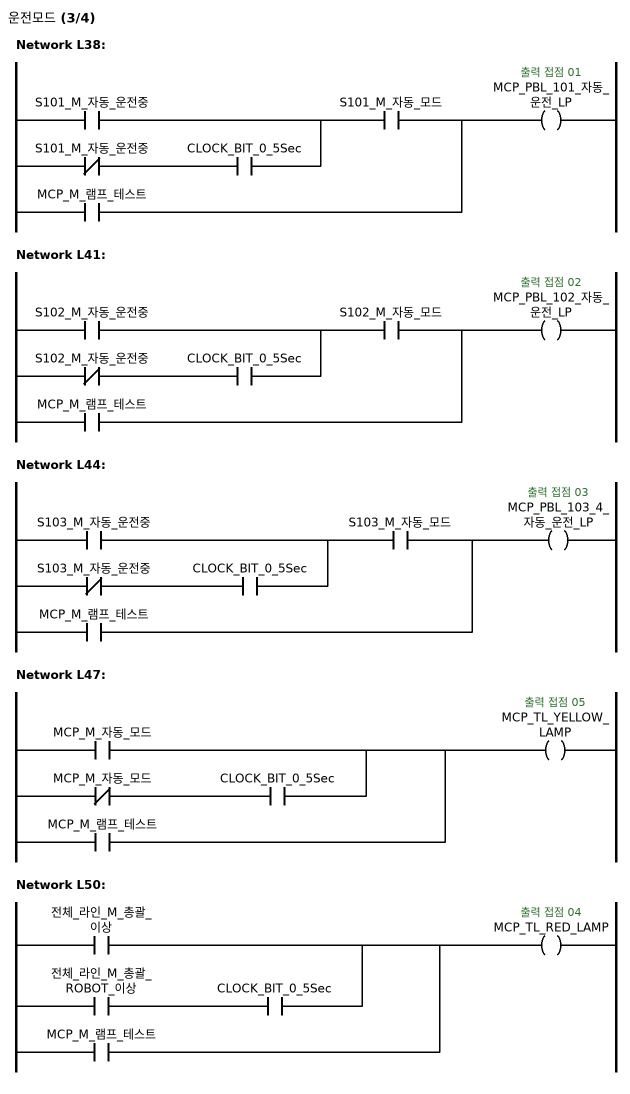
(* Rung L38 *)
MCP_PBL_101_자동_운전_LP := ((S101_M_자동_운전중 OR (NOT S101_M_자동_운전중 AND CLOCK_BIT_0_5Sec)) AND S101_M_자동_모드) OR MCP_M_램프_테스트;
(* Rung L41 *)
MCP_PBL_102_자동_운전_LP := ((S102_M_자동_운전중 OR (NOT S102_M_자동_운전중 AND CLOCK_BIT_0_5Sec)) AND S102_M_자동_모드) OR MCP_M_램프_테스트;
(* Rung L44 *)
MCP_PBL_103_4_자동_운전_LP := ((S103_M_자동_운전중 OR (NOT S103_M_자동_운전중 AND CLOCK_BIT_0_5Sec)) AND S103_M_자동_모드) OR MCP_M_램프_테스트;
(* Rung L47 *)
MCP_TL_YELLOW_LAMP := MCP_M_자동_모드 OR (NOT MCP_M_자동_모드 AND CLOCK_BIT_0_5Sec) OR MCP_M_램프_테스트;
(* Rung L50 *)
MCP_TL_RED_LAMP := 전체_라인_M_총괄_이상 OR (전체_라인_M_총괄_ROBOT_이상 AND CLOCK_BIT_0_5Sec) OR MCP_M_램프_테스트;

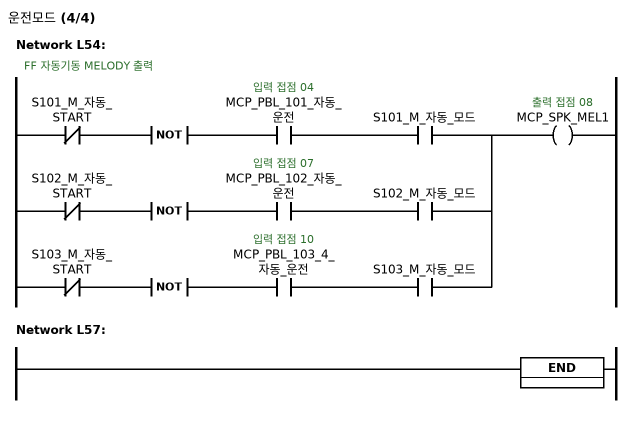
(* FF 자동기동 MELODY 출력 *)
(* Rung L54 *)
MCP_SPK_MEL1 := (S101_M_자동_START AND MCP_PBL_101_자동_운전 AND S101_M_자동_모드) OR (S102_M_자동_START AND MCP_PBL_102_자동_운전 AND S102_M_자동_모드) OR (S103_M_자동_START AND MCP_PBL_103_4_자동_운전 AND S103_M_자동_모드);
(* Rung L57 *)
END();
END_PROGRAM

PROGRAM 이상 (* task: 스캔 프로그램 *)
VAR_EXTERNAL
    AWAYS_OFF : BOOL; (* AT %MW3.0 *)
    GATE10_M_CP_TRIP : BOOL; (* AT %MW409.15 *)
    GATE10_M_GATE_OPEN : BOOL; (* AT %MW409.13 *)
    GATE10_M_비상정지 : BOOL; (* AT %MW409.7 *)
    GATE10_M_통신_이상 : BOOL; (* AT %MW409.14 *)
    GATE11_M_CP_TRIP : BOOL; (* AT %MW410.15 *)
    GATE11_M_GATE_OPEN : BOOL; (* AT %MW410.13 *)
    GATE11_M_비상정지 : BOOL; (* AT %MW410.7 *)
    GATE11_M_통신_이상 : BOOL; (* AT %MW410.14 *)
    GATE12_M_CP_TRIP : BOOL; (* AT %MW411.15 *)
    GATE12_M_GATE_OPEN : BOOL; (* AT %MW411.13 *)
    GATE12_M_비상정지 : BOOL; (* AT %MW411.7 *)
    GATE12_M_통신_이상 : BOOL; (* AT %MW411.14 *)
    MCP_DISPLAY_CP_TRIP : BOOL; (* AT %MW87632.5 *) (* 입력 접점 05 *)
    MCP_HMI_CP_TRIP : BOOL; (* AT %MW87632.4 *) (* 입력 접점 04 *)
    MCP_HUB_CP_TRIP : BOOL; (* AT %MW87632.0 *) (* 입력 접점 00 *)
    MCP_INPUT_PWR_CP_TRIP : BOOL; (* AT %MW87632.2 *) (* 입력 접점 02 *)
    MCP_MC1_OUTPUT_PWR_ON : BOOL; (* AT %MW97636.0 *) (* 출력 접점 00 *)
    MCP_M_CP_OFF_이상 : BOOL; (* AT %MW351.0 *)
    MCP_M_DISPLAY_CP_TRIP : BOOL; (* AT %MW351.6 *)
    MCP_M_HMI_CP_TRIP : BOOL; (* AT %MW351.7 *)
    MCP_M_HUB_CP_TRIP : BOOL; (* AT %MW351.1 *)
    MCP_M_INPUT_CP_TRIP : BOOL; (* AT %MW351.3 *)
    MCP_M_OUTPUT_CP_TRIP : BOOL; (* AT %MW351.4 *)
    MCP_M_OUTPUT_MC_이상 : BOOL; (* AT %MW354.8 *)
    MCP_M_PROFI_PWR_CP_TRIP : BOOL; (* AT %MW351.5 *)
    MCP_M_PS1_DC_LOW : BOOL; (* AT %MW353.6 *)
    MCP_M_PS2_DC_LOW : BOOL; (* AT %MW353.7 *)
    MCP_M_PS3_DC_LOW : BOOL; (* AT %MW353.8 *)
    MCP_M_PS4_DC_LOW : BOOL; (* AT %MW353.9 *)
    MCP_M_PS_DC_LOW : BOOL; (* AT %MW353.5 *)
    MCP_M_SAG1_1_이상 : BOOL; (* AT %MW352.1 *)
    MCP_M_SAG1_2_이상 : BOOL; (* AT %MW352.2 *)
    MCP_M_SAG_이상 : BOOL; (* AT %MW352.0 *)
    MCP_M_SPD_이상 : BOOL; (* AT %MW354.0 *)
    MCP_M_비상정지 : BOOL; (* AT %MW350.7 *)
    MCP_M_이상_리셋 : BOOL; (* AT %MW350.4 *)
    MCP_M_통신_CP_TRIP : BOOL; (* AT %MW351.2 *)
    MCP_M_통신_이상 : BOOL; (* AT %MW352.8 *)
    MCP_OUTPUT_PWR_CP_TRIP : BOOL; (* AT %MW87632.3 *) (* 입력 접점 03 *)
    MCP_PS1_DC_OK : BOOL; (* AT %MW87631.12 *) (* 입력 접점 12 *)
    MCP_PS2_DC_OK : BOOL; (* AT %MW87631.13 *) (* 입력 접점 13 *)
    MCP_PS3_DC_OK : BOOL; (* AT %MW87631.14 *) (* 입력 접점 14 *)
    MCP_SAFTY_MC_ON : BOOL; (* AT %MW87632.9 *) (* 입력 접점 09 *)
    MCP_통신_CP_TRIP : BOOL; (* AT %MW87632.1 *) (* 입력 접점 01 *)
    PWR_SAG1_DSUB1_NOMAL1 : BOOL; (* AT %MW87631.10 *) (* 입력 접점 10 *)
    PWR_SAG1_DSUB8_NOMAL2 : BOOL; (* AT %MW87631.11 *) (* 입력 접점 11 *)
    PWR_SPD1_NOMAL : BOOL; (* AT %MW87631.8 *) (* 입력 접점 08 *)
    S101_M_총괄_CP_이상 : BOOL; (* AT %MW1009.7 *)
    S101_M_총괄_CT_이상 : BOOL; (* AT %MW1010.4 *)
    S101_M_총괄_EOCR_이상 : BOOL; (* AT %MW1009.8 *)
    S101_M_총괄_INV_이상 : BOOL; (* AT %MW1009.9 *)
    S101_M_총괄_LS_이상 : BOOL; (* AT %MW1009.15 *)
    S101_M_총괄_MATCH_이상 : BOOL; (* AT %MW1010.0 *)
    S101_M_총괄_MC_이상 : BOOL; (* AT %MW1009.13 *)
    S101_M_총괄_MOTOR_이상 : BOOL; (* AT %MW1010.3 *)
    S101_M_총괄_NFB_이상 : BOOL; (* AT %MW1009.11 *)
    S101_M_총괄_ROBOT_이상 : BOOL; (* AT %MW1010.1 *)
    S101_M_총괄_SAFETY_이상 : BOOL; (* AT %MW1009.2 *)
    S101_M_총괄_SRV_이상 : BOOL; (* AT %MW1009.10 *)
    S101_M_총괄_공기압_이상 : BOOL; (* AT %MW1009.3 *)
    S101_M_총괄_비상정지_이상 : BOOL; (* AT %MW1009.1 *)
    S101_M_총괄_사양_이상 : BOOL; (* AT %MW1009.6 *)
    S101_M_총괄_오버런_이상 : BOOL; (* AT %MW1009.12 *)
    S101_M_총괄_용점타점수_이상 : BOOL; (* AT %MW1010.2 *)
    S101_M_총괄_제품감지_이상 : BOOL; (* AT %MW1009.4 *)
    S101_M_총괄_차종_이상 : BOOL; (* AT %MW1009.5 *)
    S101_M_총괄_통신_이상 : BOOL; (* AT %MW1009.14 *)
    S102_M_총괄_CP_이상 : BOOL; (* AT %MW1509.7 *)
    S102_M_총괄_CT_이상 : BOOL; (* AT %MW1510.4 *)
    S102_M_총괄_EOCR_이상 : BOOL; (* AT %MW1509.8 *)
    S102_M_총괄_INV_이상 : BOOL; (* AT %MW1509.9 *)
    S102_M_총괄_LS_이상 : BOOL; (* AT %MW1509.15 *)
    S102_M_총괄_MATCH_이상 : BOOL; (* AT %MW1510.0 *)
    S102_M_총괄_MC_이상 : BOOL; (* AT %MW1509.13 *)
    S102_M_총괄_MOTOR_이상 : BOOL; (* AT %MW1510.3 *)
    S102_M_총괄_NFB_이상 : BOOL; (* AT %MW1509.11 *)
    S102_M_총괄_ROBOT_이상 : BOOL; (* AT %MW1510.1 *)
    S102_M_총괄_SAFETY_이상 : BOOL; (* AT %MW1509.2 *)
    S102_M_총괄_SRV_이상 : BOOL; (* AT %MW1509.10 *)
    S102_M_총괄_공기압_이상 : BOOL; (* AT %MW1509.3 *)
    S102_M_총괄_비상정지_이상 : BOOL; (* AT %MW1509.1 *)
    S102_M_총괄_사양_이상 : BOOL; (* AT %MW1509.6 *)
    S102_M_총괄_오버런_이상 : BOOL; (* AT %MW1509.12 *)
    S102_M_총괄_용점타점수_이상 : BOOL; (* AT %MW1510.2 *)
    S102_M_총괄_이상 : BOOL; (* AT %MW1509.0 *)
    S102_M_총괄_제품감지_이상 : BOOL; (* AT %MW1509.4 *)
    S102_M_총괄_차종_이상 : BOOL; (* AT %MW1509.5 *)
    S102_M_총괄_통신_이상 : BOOL; (* AT %MW1509.14 *)
    S103_M_총괄_CP_이상 : BOOL; (* AT %MW2009.7 *)
    S103_M_총괄_CT_이상 : BOOL; (* AT %MW2010.4 *)
    S103_M_총괄_EOCR_이상 : BOOL; (* AT %MW2009.8 *)
    S103_M_총괄_INV_이상 : BOOL; (* AT %MW2009.9 *)
    S103_M_총괄_LS_이상 : BOOL; (* AT %MW2009.15 *)
    S103_M_총괄_MATCH_이상 : BOOL; (* AT %MW2010.0 *)
    S103_M_총괄_MC_이상 : BOOL; (* AT %MW2009.13 *)
    S103_M_총괄_MOTOR_이상 : BOOL; (* AT %MW2010.3 *)
    S103_M_총괄_NFB_이상 : BOOL; (* AT %MW2009.11 *)
    S103_M_총괄_ROBOT_이상 : BOOL; (* AT %MW2010.1 *)
    S103_M_총괄_SAFETY_이상 : BOOL; (* AT %MW2009.2 *)
    S103_M_총괄_SRV_이상 : BOOL; (* AT %MW2009.10 *)
    S103_M_총괄_공기압_이상 : BOOL; (* AT %MW2009.3 *)
    S103_M_총괄_비상정지_이상 : BOOL; (* AT %MW2009.1 *)
    S103_M_총괄_사양_이상 : BOOL; (* AT %MW2009.6 *)
    S103_M_총괄_오버런_이상 : BOOL; (* AT %MW2009.12 *)
    S103_M_총괄_용점타점수_이상 : BOOL; (* AT %MW2010.2 *)
    S103_M_총괄_이상 : BOOL; (* AT %MW2009.0 *)
    S103_M_총괄_제품감지_이상 : BOOL; (* AT %MW2009.4 *)
    S103_M_총괄_차종_이상 : BOOL; (* AT %MW2009.5 *)
    S103_M_총괄_통신_이상 : BOOL; (* AT %MW2009.14 *)
    S104_M_총괄_CP_이상 : BOOL; (* AT %MW2509.7 *)
    S104_M_총괄_CT_이상 : BOOL; (* AT %MW2510.4 *)
    S104_M_총괄_EOCR_이상 : BOOL; (* AT %MW2509.8 *)
    S104_M_총괄_INV_이상 : BOOL; (* AT %MW2509.9 *)
    S104_M_총괄_LS_이상 : BOOL; (* AT %MW2509.15 *)
    S104_M_총괄_MATCH_이상 : BOOL; (* AT %MW2510.0 *)
    S104_M_총괄_MC_이상 : BOOL; (* AT %MW2509.13 *)
    S104_M_총괄_MOTOR_이상 : BOOL; (* AT %MW2510.3 *)
    S104_M_총괄_NFB_이상 : BOOL; (* AT %MW2509.11 *)
    S104_M_총괄_ROBOT_이상 : BOOL; (* AT %MW2510.1 *)
    S104_M_총괄_SAFETY_이상 : BOOL; (* AT %MW2509.2 *)
    S104_M_총괄_SRV_이상 : BOOL; (* AT %MW2509.10 *)
    S104_M_총괄_공기압_이상 : BOOL; (* AT %MW2509.3 *)
    S104_M_총괄_비상정지_이상 : BOOL; (* AT %MW2509.1 *)
    S104_M_총괄_사양_이상 : BOOL; (* AT %MW2509.6 *)
    S104_M_총괄_오버런_이상 : BOOL; (* AT %MW2509.12 *)
    S104_M_총괄_용점타점수_이상 : BOOL; (* AT %MW2510.2 *)
    S104_M_총괄_제품감지_이상 : BOOL; (* AT %MW2509.4 *)
    S104_M_총괄_차종_이상 : BOOL; (* AT %MW2509.5 *)
    S104_M_총괄_통신_이상 : BOOL; (* AT %MW2509.14 *)
    SRV1_M_PS1_DC_LOW : BOOL; (* AT %MW357.2 *)
    SRV1_M_PS2_DC_LOW : BOOL; (* AT %MW357.3 *)
    SRV1_M_SPD_이상 : BOOL; (* AT %MW357.1 *)
    SRV1_M_총괄_이상 : BOOL; (* AT %MW357.0 *)
    SRV1_M_통신_이상 : BOOL; (* AT %MW356.4 *)
    SRV_PNL_CP_ON : BOOL; (* AT %MW85363.15 *)
    SRV_PNL_PS_NOMAL : BOOL; (* AT %MW85363.12 *)
    SRV_PNL_SPD_NOMAL : BOOL; (* AT %MW85203.9 *)
    _0005_EB20_CFG_ER : BOOL; (* AT %MW185124.0 *) (* EB 구성 에러 *)
    _0005_EB20_DEER : BOOL; (* AT %MW185124.1 *) (* EB 운전 중 탈락 *)
    _0005_EB20_IO_DEER : BOOL; (* AT %MW185125.2 *) (* EB IO 탈락 에러 *)
    _0005_EB20_IO_TYER : BOOL; (* AT %MW185125.1 *) (* EB IO 타입 에러 *)
    _0007_EB63_CFG_ER : BOOL; (* AT %MW187040.0 *) (* EB 구성 에러 *)
    _0007_EB63_DEER : BOOL; (* AT %MW187040.1 *) (* EB 운전 중 탈락 *)
    _0007_EB63_IO_DEER : BOOL; (* AT %MW187041.2 *) (* EB IO 탈락 에러 *)
    _0007_EB63_IO_TYER : BOOL; (* AT %MW187041.1 *) (* EB IO 타입 에러 *)
    전체_M_이상_리셋 : BOOL; (* AT %MW308.2 *) (* 전체 M 이상 리셋 *)
    전체_라인_M_총괄_CP_OFF : BOOL; (* AT %MW300.7 *)
    전체_라인_M_총괄_CT_이상 : BOOL; (* AT %MW301.4 *)
    전체_라인_M_총괄_EOCR_이상 : BOOL; (* AT %MW300.8 *)
    전체_라인_M_총괄_GATE_OPEN_이상 : BOOL; (* AT %MW301.5 *)
    전체_라인_M_총괄_INV_이상 : BOOL; (* AT %MW300.9 *)
    전체_라인_M_총괄_LS_이상 : BOOL; (* AT %MW300.15 *)
    전체_라인_M_총괄_MATCH_이상 : BOOL; (* AT %MW301.0 *)
    전체_라인_M_총괄_MC_이상 : BOOL; (* AT %MW300.13 *)
    전체_라인_M_총괄_MOTOR_이상 : BOOL; (* AT %MW301.3 *)
    전체_라인_M_총괄_NFB_이상 : BOOL; (* AT %MW300.11 *)
    전체_라인_M_총괄_PS_DC_LOW : BOOL; (* AT %MW301.7 *)
    전체_라인_M_총괄_ROBOT_이상 : BOOL; (* AT %MW301.1 *)
    전체_라인_M_총괄_SAFETY_이상 : BOOL; (* AT %MW300.2 *)
    전체_라인_M_총괄_SAG_이상 : BOOL; (* AT %MW301.6 *)
    전체_라인_M_총괄_SPD_이상 : BOOL; (* AT %MW301.8 *)
    전체_라인_M_총괄_SRV_이상 : BOOL; (* AT %MW300.10 *)
    전체_라인_M_총괄_공기압_이상 : BOOL; (* AT %MW300.3 *)
    전체_라인_M_총괄_비상정지_이상 : BOOL; (* AT %MW300.1 *)
    전체_라인_M_총괄_사양_이상 : BOOL; (* AT %MW300.6 *)
    전체_라인_M_총괄_오버런_이상 : BOOL; (* AT %MW300.12 *)
    전체_라인_M_총괄_용점타점수_이상 : BOOL; (* AT %MW301.2 *)
    전체_라인_M_총괄_이상 : BOOL; (* AT %MW300.0 *)
    전체_라인_M_총괄_제품감지_이상 : BOOL; (* AT %MW300.4 *)
    전체_라인_M_총괄_차종_이상 : BOOL; (* AT %MW300.5 *)
    전체_라인_M_총괄_통신_이상 : BOOL; (* AT %MW300.14 *)
END_VAR
VAR
    INST1 : TON;
    INST10 : TON;
    INST11 : TON;
    INST12 : TON;
    INST13 : TON;
    INST14 : TON;
    INST15 : TON;
    INST2 : TON;
    INST24 : TON;
    INST25 : TON;
    INST26 : TON;
    INST27 : TON;
    INST3 : TON;
    INST4 : TON;
    INST5 : TON;
    INST6 : TON;
    INST7 : TON;
    INST8 : TON;
    INST9 : TON;
END_VAR

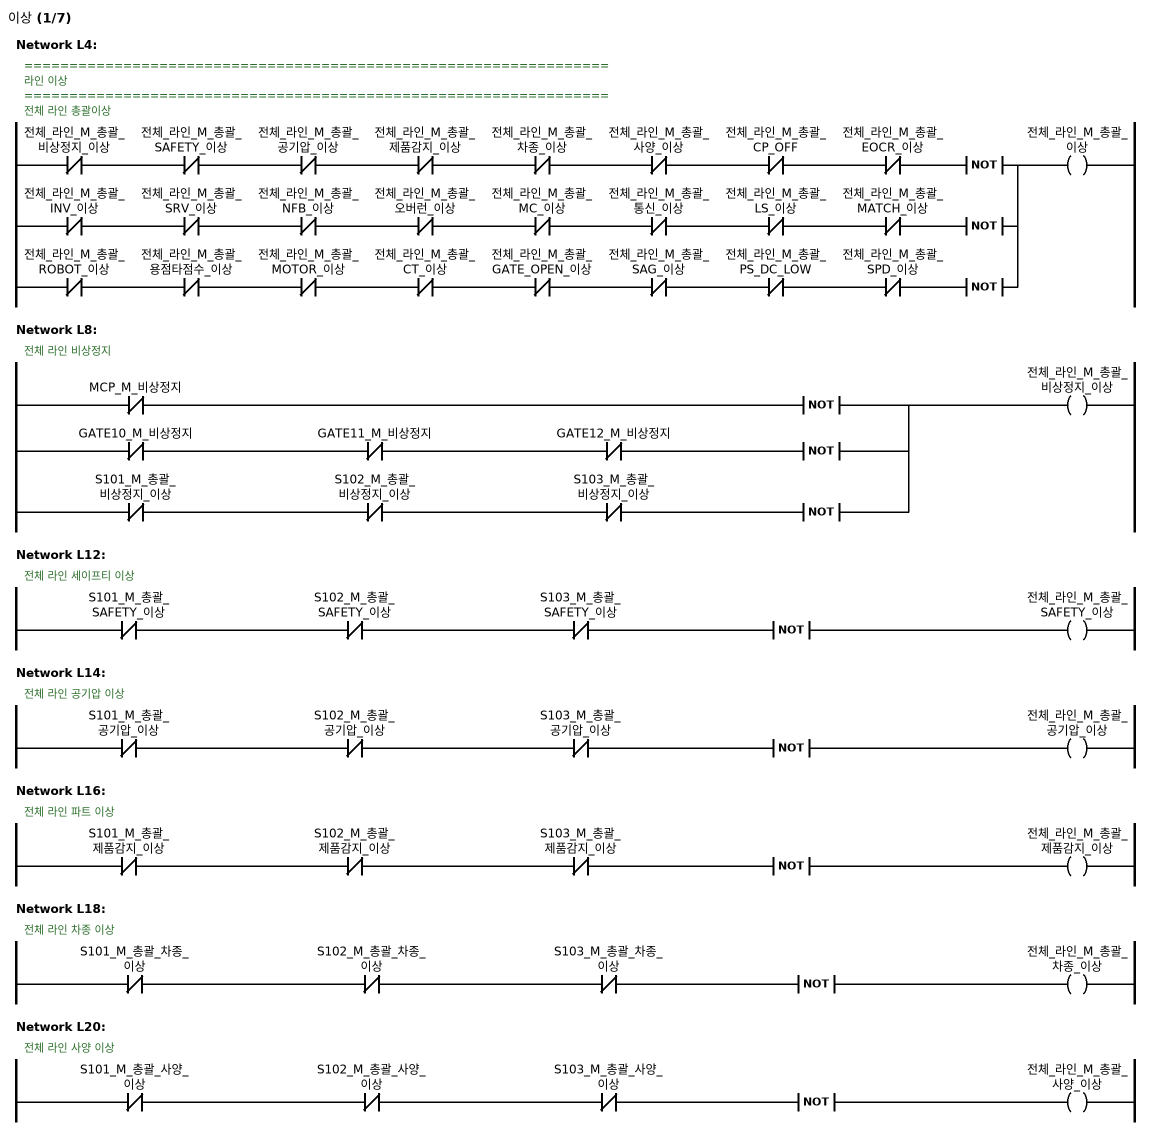
(* ================================================================= *)
(* 라인 이상 *)
(* ================================================================= *)
(* 전체 라인 총괄이상 *)
(* Rung L4 *)
전체_라인_M_총괄_이상 := NOT (NOT 전체_라인_M_총괄_비상정지_이상 AND NOT 전체_라인_M_총괄_SAFETY_이상 AND NOT 전체_라인_M_총괄_공기압_이상 AND NOT 전체_라인_M_총괄_제품감지_이상 AND NOT 전체_라인_M_총괄_차종_이상 AND NOT 전체_라인_M_총괄_사양_이상 AND NOT 전체_라인_M_총괄_CP_OFF AND NOT 전체_라인_M_총괄_EOCR_이상) OR NOT (NOT 전체_라인_M_총괄_INV_이상 AND NOT 전체_라인_M_총괄_SRV_이상 AND NOT 전체_라인_M_총괄_NFB_이상 AND NOT 전체_라인_M_총괄_오버런_이상 AND NOT 전체_라인_M_총괄_MC_이상 AND NOT 전체_라인_M_총괄_통신_이상 AND NOT 전체_라인_M_총괄_LS_이상 AND NOT 전체_라인_M_총괄_MATCH_이상) OR NOT (NOT 전체_라인_M_총괄_ROBOT_이상 AND NOT 전체_라인_M_총괄_용점타점수_이상 AND NOT 전체_라인_M_총괄_MOTOR_이상 AND NOT 전체_라인_M_총괄_CT_이상 AND NOT 전체_라인_M_총괄_GATE_OPEN_이상 AND NOT 전체_라인_M_총괄_SAG_이상 AND NOT 전체_라인_M_총괄_PS_DC_LOW AND NOT 전체_라인_M_총괄_SPD_이상);
(* 전체 라인 비상정지 *)
(* Rung L8 *)
전체_라인_M_총괄_비상정지_이상 := MCP_M_비상정지 OR NOT (NOT GATE10_M_비상정지 AND NOT GATE11_M_비상정지 AND NOT GATE12_M_비상정지) OR NOT (NOT S101_M_총괄_비상정지_이상 AND NOT S102_M_총괄_비상정지_이상 AND NOT S103_M_총괄_비상정지_이상);
(* 전체 라인 세이프티 이상 *)
(* Rung L12 *)
전체_라인_M_총괄_SAFETY_이상 := NOT (NOT S101_M_총괄_SAFETY_이상 AND NOT S102_M_총괄_SAFETY_이상 AND NOT S103_M_총괄_SAFETY_이상);
(* 전체 라인 공기압 이상 *)
(* Rung L14 *)
전체_라인_M_총괄_공기압_이상 := NOT (NOT S101_M_총괄_공기압_이상 AND NOT S102_M_총괄_공기압_이상 AND NOT S103_M_총괄_공기압_이상);
(* 전체 라인 파트 이상 *)
(* Rung L16 *)
전체_라인_M_총괄_제품감지_이상 := NOT (NOT S101_M_총괄_제품감지_이상 AND NOT S102_M_총괄_제품감지_이상 AND NOT S103_M_총괄_제품감지_이상);
(* 전체 라인 차종 이상 *)
(* Rung L18 *)
전체_라인_M_총괄_차종_이상 := NOT (NOT S101_M_총괄_차종_이상 AND NOT S102_M_총괄_차종_이상 AND NOT S103_M_총괄_차종_이상);
(* 전체 라인 사양 이상 *)
(* Rung L20 *)
전체_라인_M_총괄_사양_이상 := NOT (NOT S101_M_총괄_사양_이상 AND NOT S102_M_총괄_사양_이상 AND NOT S103_M_총괄_사양_이상);

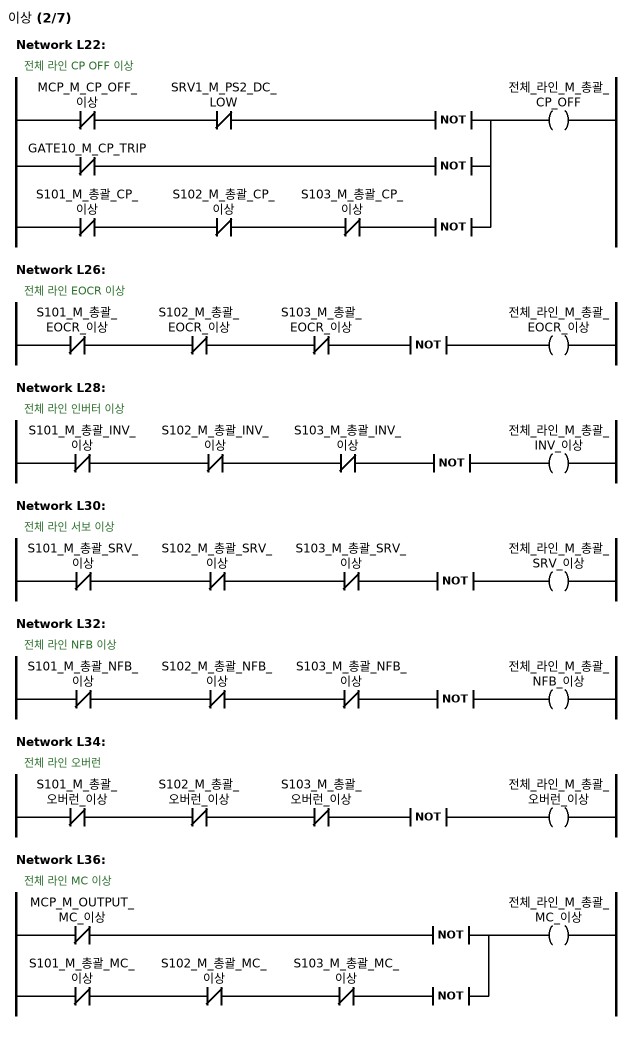
(* 전체 라인 CP OFF 이상 *)
(* Rung L22 *)
전체_라인_M_총괄_CP_OFF := NOT (NOT MCP_M_CP_OFF_이상 AND NOT SRV1_M_PS2_DC_LOW) OR GATE10_M_CP_TRIP OR NOT (NOT S101_M_총괄_CP_이상 AND NOT S102_M_총괄_CP_이상 AND NOT S103_M_총괄_CP_이상);
(* 전체 라인 EOCR 이상 *)
(* Rung L26 *)
전체_라인_M_총괄_EOCR_이상 := NOT (NOT S101_M_총괄_EOCR_이상 AND NOT S102_M_총괄_EOCR_이상 AND NOT S103_M_총괄_EOCR_이상);
(* 전체 라인 인버터 이상 *)
(* Rung L28 *)
전체_라인_M_총괄_INV_이상 := NOT (NOT S101_M_총괄_INV_이상 AND NOT S102_M_총괄_INV_이상 AND NOT S103_M_총괄_INV_이상);
(* 전체 라인 서보 이상 *)
(* Rung L30 *)
전체_라인_M_총괄_SRV_이상 := NOT (NOT S101_M_총괄_SRV_이상 AND NOT S102_M_총괄_SRV_이상 AND NOT S103_M_총괄_SRV_이상);
(* 전체 라인 NFB 이상 *)
(* Rung L32 *)
전체_라인_M_총괄_NFB_이상 := NOT (NOT S101_M_총괄_NFB_이상 AND NOT S102_M_총괄_NFB_이상 AND NOT S103_M_총괄_NFB_이상);
(* 전체 라인 오버런 *)
(* Rung L34 *)
전체_라인_M_총괄_오버런_이상 := NOT (NOT S101_M_총괄_오버런_이상 AND NOT S102_M_총괄_오버런_이상 AND NOT S103_M_총괄_오버런_이상);
(* 전체 라인 MC 이상 *)
(* Rung L36 *)
전체_라인_M_총괄_MC_이상 := MCP_M_OUTPUT_MC_이상 OR NOT (NOT S101_M_총괄_MC_이상 AND NOT S102_M_총괄_MC_이상 AND NOT S103_M_총괄_MC_이상);

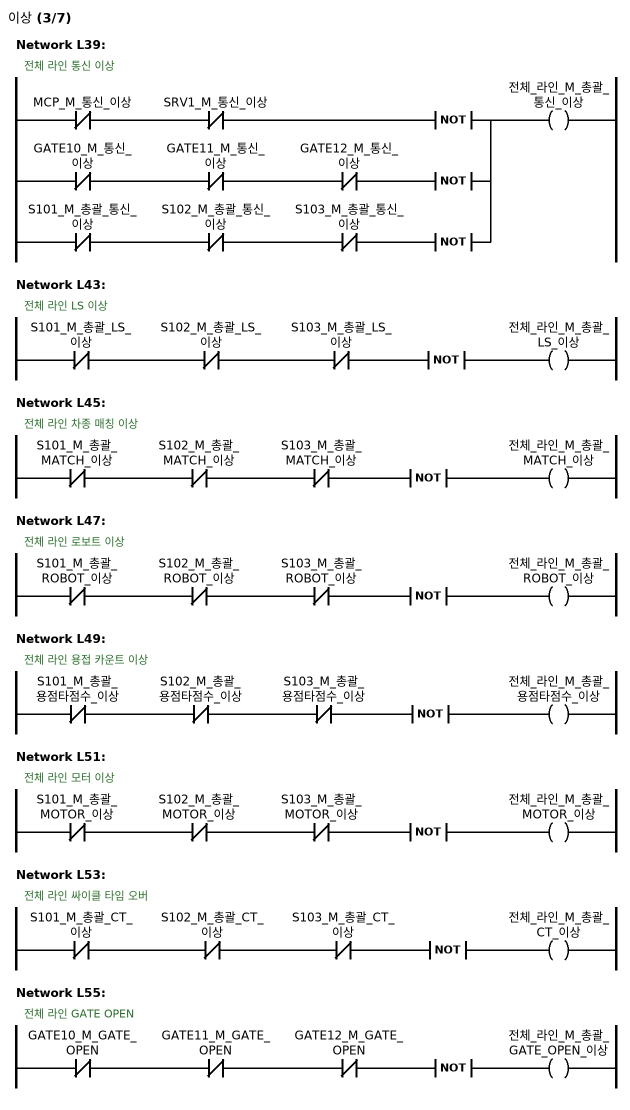
(* 전체 라인 통신 이상 *)
(* Rung L39 *)
전체_라인_M_총괄_통신_이상 := NOT (NOT MCP_M_통신_이상 AND NOT SRV1_M_통신_이상) OR NOT (NOT GATE10_M_통신_이상 AND NOT GATE11_M_통신_이상 AND NOT GATE12_M_통신_이상) OR NOT (NOT S101_M_총괄_통신_이상 AND NOT S102_M_총괄_통신_이상 AND NOT S103_M_총괄_통신_이상);
(* 전체 라인 LS 이상 *)
(* Rung L43 *)
전체_라인_M_총괄_LS_이상 := NOT (NOT S101_M_총괄_LS_이상 AND NOT S102_M_총괄_LS_이상 AND NOT S103_M_총괄_LS_이상);
(* 전체 라인 차종 매칭 이상 *)
(* Rung L45 *)
전체_라인_M_총괄_MATCH_이상 := NOT (NOT S101_M_총괄_MATCH_이상 AND NOT S102_M_총괄_MATCH_이상 AND NOT S103_M_총괄_MATCH_이상);
(* 전체 라인 로보트 이상 *)
(* Rung L47 *)
전체_라인_M_총괄_ROBOT_이상 := NOT (NOT S101_M_총괄_ROBOT_이상 AND NOT S102_M_총괄_ROBOT_이상 AND NOT S103_M_총괄_ROBOT_이상);
(* 전체 라인 용접 카운트 이상 *)
(* Rung L49 *)
전체_라인_M_총괄_용점타점수_이상 := NOT (NOT S101_M_총괄_용점타점수_이상 AND NOT S102_M_총괄_용점타점수_이상 AND NOT S103_M_총괄_용점타점수_이상);
(* 전체 라인 모터 이상 *)
(* Rung L51 *)
전체_라인_M_총괄_MOTOR_이상 := NOT (NOT S101_M_총괄_MOTOR_이상 AND NOT S102_M_총괄_MOTOR_이상 AND NOT S103_M_총괄_MOTOR_이상);
(* 전체 라인 싸이클 타임 오버 *)
(* Rung L53 *)
전체_라인_M_총괄_CT_이상 := NOT (NOT S101_M_총괄_CT_이상 AND NOT S102_M_총괄_CT_이상 AND NOT S103_M_총괄_CT_이상);
(* 전체 라인 GATE OPEN *)
(* Rung L55 *)
전체_라인_M_총괄_GATE_OPEN_이상 := NOT (NOT GATE10_M_GATE_OPEN AND NOT GATE11_M_GATE_OPEN AND NOT GATE12_M_GATE_OPEN);

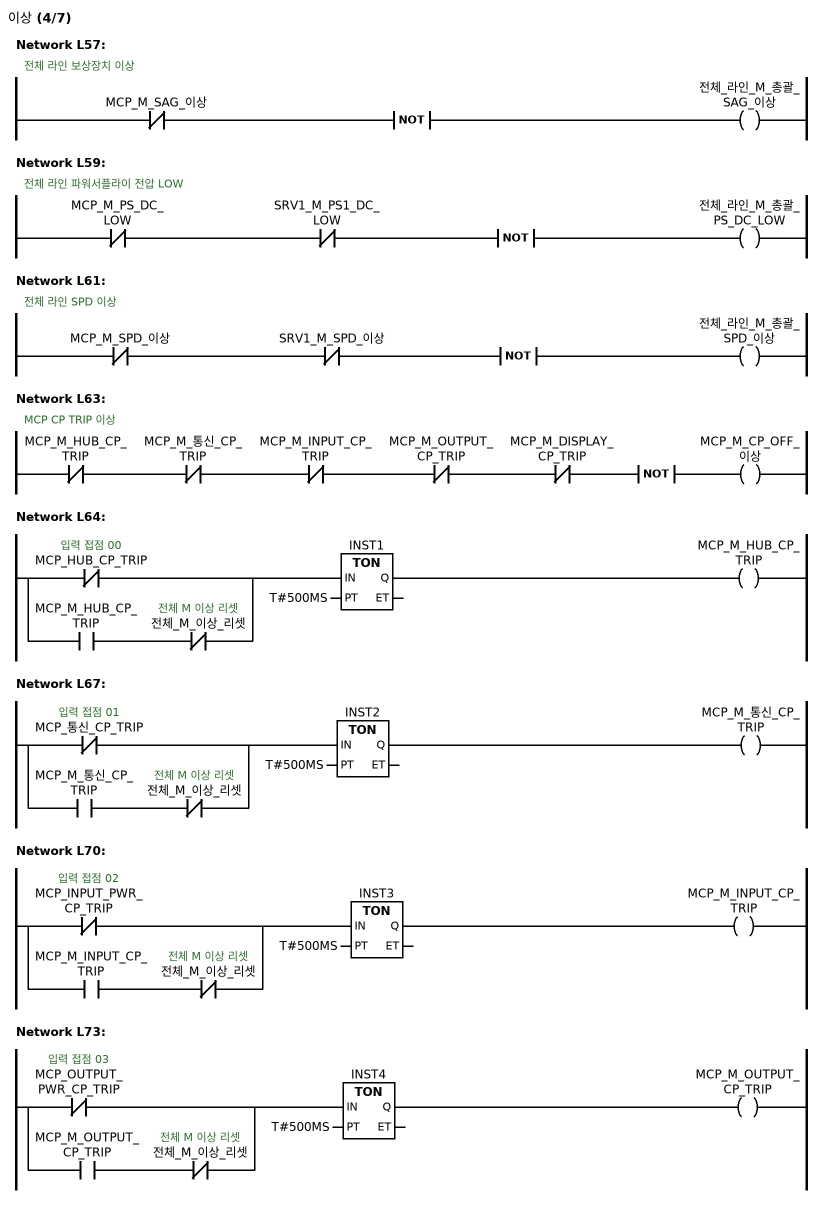
(* 전체 라인 보상장치 이상 *)
(* Rung L57 *)
전체_라인_M_총괄_SAG_이상 := MCP_M_SAG_이상;
(* 전체 라인 파워서플라이 전압 LOW *)
(* Rung L59 *)
전체_라인_M_총괄_PS_DC_LOW := NOT (NOT MCP_M_PS_DC_LOW AND NOT SRV1_M_PS1_DC_LOW);
(* 전체 라인 SPD 이상 *)
(* Rung L61 *)
전체_라인_M_총괄_SPD_이상 := NOT (NOT MCP_M_SPD_이상 AND NOT SRV1_M_SPD_이상);
(* MCP CP TRIP 이상 *)
(* Rung L63 *)
MCP_M_CP_OFF_이상 := NOT (NOT MCP_M_HUB_CP_TRIP AND NOT MCP_M_통신_CP_TRIP AND NOT MCP_M_INPUT_CP_TRIP AND NOT MCP_M_OUTPUT_CP_TRIP AND NOT MCP_M_DISPLAY_CP_TRIP);
(* Rung L64 *)
INST1(IN := NOT MCP_HUB_CP_TRIP OR (MCP_M_HUB_CP_TRIP AND NOT 전체_M_이상_리셋), PT := T#500MS);
MCP_M_HUB_CP_TRIP := INST1.Q;
(* Rung L67 *)
INST2(IN := NOT MCP_통신_CP_TRIP OR (MCP_M_통신_CP_TRIP AND NOT 전체_M_이상_리셋), PT := T#500MS);
MCP_M_통신_CP_TRIP := INST2.Q;
(* Rung L70 *)
INST3(IN := NOT MCP_INPUT_PWR_CP_TRIP OR (MCP_M_INPUT_CP_TRIP AND NOT 전체_M_이상_리셋), PT := T#500MS);
MCP_M_INPUT_CP_TRIP := INST3.Q;
(* Rung L73 *)
INST4(IN := NOT MCP_OUTPUT_PWR_CP_TRIP OR (MCP_M_OUTPUT_CP_TRIP AND NOT 전체_M_이상_리셋), PT := T#500MS);
MCP_M_OUTPUT_CP_TRIP := INST4.Q;

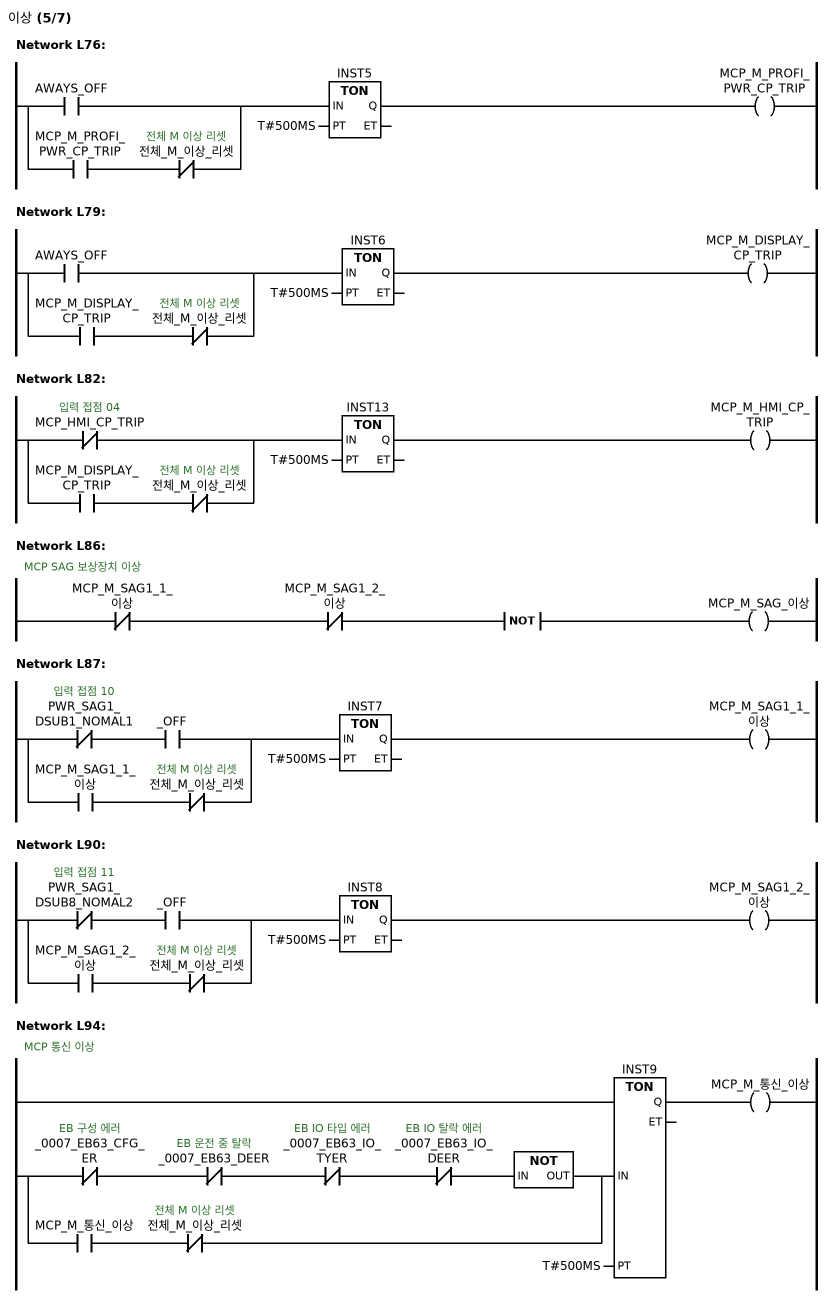
(* Rung L76 *)
INST5(IN := AWAYS_OFF OR (MCP_M_PROFI_PWR_CP_TRIP AND NOT 전체_M_이상_리셋), PT := T#500MS);
MCP_M_PROFI_PWR_CP_TRIP := INST5.Q;
(* Rung L79 *)
INST6(IN := AWAYS_OFF OR (MCP_M_DISPLAY_CP_TRIP AND NOT 전체_M_이상_리셋), PT := T#500MS);
MCP_M_DISPLAY_CP_TRIP := INST6.Q;
(* Rung L82 *)
INST13(IN := NOT MCP_HMI_CP_TRIP OR (MCP_M_DISPLAY_CP_TRIP AND NOT 전체_M_이상_리셋), PT := T#500MS);
MCP_M_HMI_CP_TRIP := INST13.Q;
(* MCP SAG 보상장치 이상 *)
(* Rung L86 *)
MCP_M_SAG_이상 := NOT (NOT MCP_M_SAG1_1_이상 AND NOT MCP_M_SAG1_2_이상);
(* Rung L87 *)
INST7(IN := (NOT PWR_SAG1_DSUB1_NOMAL1 AND _OFF) OR (MCP_M_SAG1_1_이상 AND NOT 전체_M_이상_리셋), PT := T#500MS);
MCP_M_SAG1_1_이상 := INST7.Q;
(* Rung L90 *)
INST8(IN := (NOT PWR_SAG1_DSUB8_NOMAL2 AND _OFF) OR (MCP_M_SAG1_2_이상 AND NOT 전체_M_이상_리셋), PT := T#500MS);
MCP_M_SAG1_2_이상 := INST8.Q;
(* MCP 통신 이상 *)
(* Rung L94 *)
INST9(IN := (NOT (NOT _0007_EB63_CFG_ER AND NOT _0007_EB63_DEER AND NOT _0007_EB63_IO_TYER AND NOT _0007_EB63_IO_DEER)) OR (MCP_M_통신_이상 AND NOT 전체_M_이상_리셋), PT := T#500MS);
MCP_M_통신_이상 := INST9.Q;

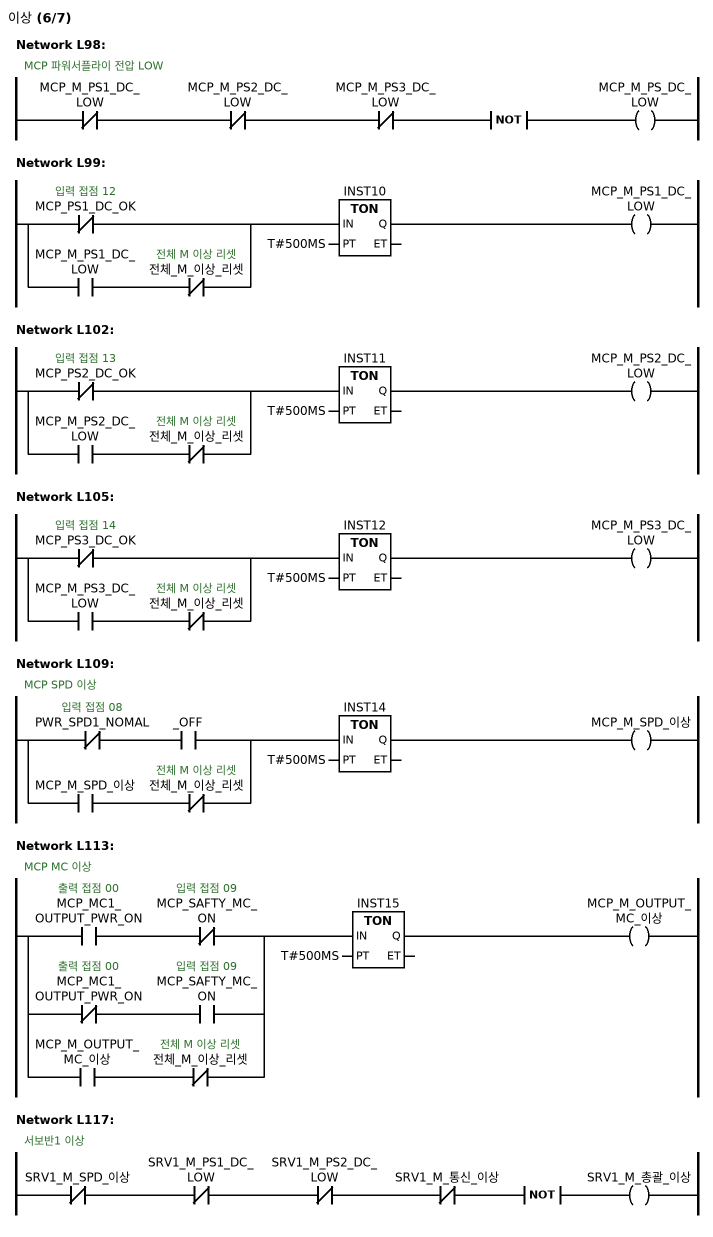
(* MCP 파워서플라이 전압 LOW *)
(* Rung L98 *)
MCP_M_PS_DC_LOW := NOT (NOT MCP_M_PS1_DC_LOW AND NOT MCP_M_PS2_DC_LOW AND NOT MCP_M_PS3_DC_LOW);
(* Rung L99 *)
INST10(IN := NOT MCP_PS1_DC_OK OR (MCP_M_PS1_DC_LOW AND NOT 전체_M_이상_리셋), PT := T#500MS);
MCP_M_PS1_DC_LOW := INST10.Q;
(* Rung L102 *)
INST11(IN := NOT MCP_PS2_DC_OK OR (MCP_M_PS2_DC_LOW AND NOT 전체_M_이상_리셋), PT := T#500MS);
MCP_M_PS2_DC_LOW := INST11.Q;
(* Rung L105 *)
INST12(IN := NOT MCP_PS3_DC_OK OR (MCP_M_PS3_DC_LOW AND NOT 전체_M_이상_리셋), PT := T#500MS);
MCP_M_PS3_DC_LOW := INST12.Q;
(* MCP SPD 이상 *)
(* Rung L109 *)
INST14(IN := (NOT PWR_SPD1_NOMAL AND _OFF) OR (MCP_M_SPD_이상 AND NOT 전체_M_이상_리셋), PT := T#500MS);
MCP_M_SPD_이상 := INST14.Q;
(* MCP MC 이상 *)
(* Rung L113 *)
INST15(IN := (MCP_MC1_OUTPUT_PWR_ON AND NOT MCP_SAFTY_MC_ON) OR (NOT MCP_MC1_OUTPUT_PWR_ON AND MCP_SAFTY_MC_ON) OR (MCP_M_OUTPUT_MC_이상 AND NOT 전체_M_이상_리셋), PT := T#500MS);
MCP_M_OUTPUT_MC_이상 := INST15.Q;
(* 서보반1 이상 *)
(* Rung L117 *)
SRV1_M_총괄_이상 := NOT (NOT SRV1_M_SPD_이상 AND NOT SRV1_M_PS1_DC_LOW AND NOT SRV1_M_PS2_DC_LOW AND NOT SRV1_M_통신_이상);

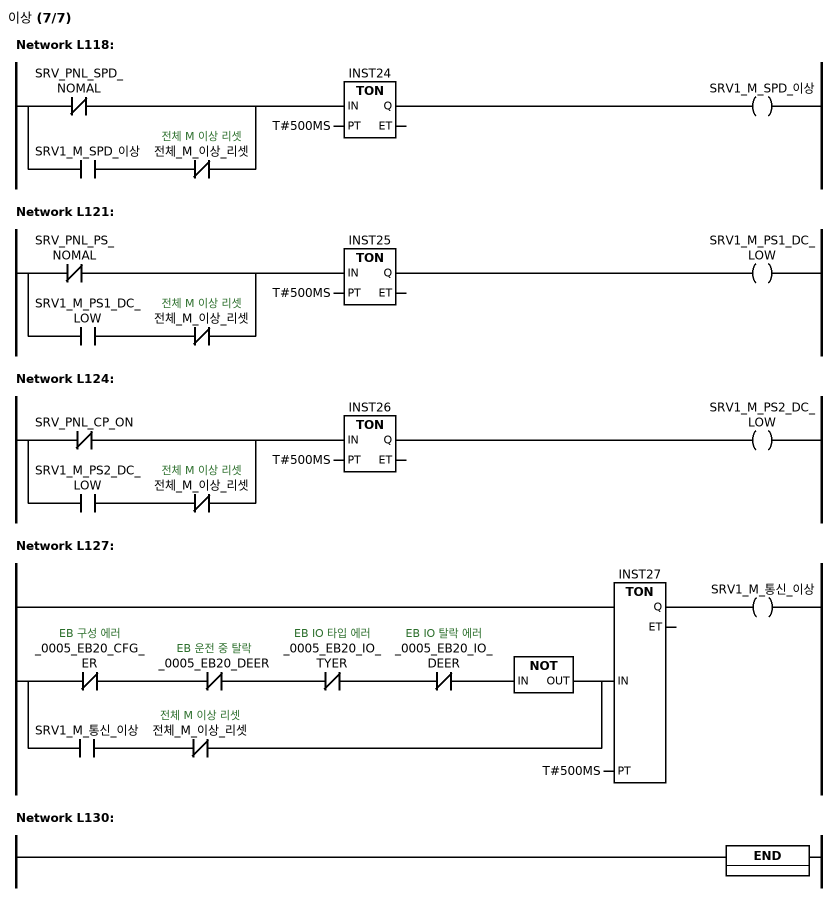
(* Rung L118 *)
INST24(IN := NOT SRV_PNL_SPD_NOMAL OR (SRV1_M_SPD_이상 AND NOT 전체_M_이상_리셋), PT := T#500MS);
SRV1_M_SPD_이상 := INST24.Q;
(* Rung L121 *)
INST25(IN := NOT SRV_PNL_PS_NOMAL OR (SRV1_M_PS1_DC_LOW AND NOT 전체_M_이상_리셋), PT := T#500MS);
SRV1_M_PS1_DC_LOW := INST25.Q;
(* Rung L124 *)
INST26(IN := NOT SRV_PNL_CP_ON OR (SRV1_M_PS2_DC_LOW AND NOT 전체_M_이상_리셋), PT := T#500MS);
SRV1_M_PS2_DC_LOW := INST26.Q;
(* Rung L127 *)
INST27(IN := (NOT (NOT _0005_EB20_CFG_ER AND NOT _0005_EB20_DEER AND NOT _0005_EB20_IO_TYER AND NOT _0005_EB20_IO_DEER)) OR (SRV1_M_통신_이상 AND NOT 전체_M_이상_리셋), PT := T#500MS);
SRV1_M_통신_이상 := INST27.Q;
(* Rung L130 *)
END();
END_PROGRAM

PROGRAM OP (* task: 스캔 프로그램 *)
VAR_EXTERNAL
    AWAYS_OFF : BOOL; (* AT %MW3.0 *)
    CLOCK_BIT_0_5Sec : BOOL; (* AT %MW0.3 *)
    GATE10_M_CP_TRIP : BOOL; (* AT %MW409.15 *)
    GATE10_M_RESTART : BOOL; (* AT %MW409.1 *)
    GATE10_M_도어_잠김 : BOOL; (* AT %MW409.3 *)
    GATE10_M_비상정지 : BOOL; (* AT %MW409.7 *)
    GATE10_M_이상_리셋 : BOOL; (* AT %MW409.0 *)
    GATE10_M_정상 : BOOL; (* AT %MW409.4 *)
    GATE10_M_정지_CALL : BOOL; (* AT %MW409.2 *)
    GATE10_M_통신_이상 : BOOL; (* AT %MW409.14 *)
    GATE11_M_CP_TRIP : BOOL; (* AT %MW410.15 *)
    GATE11_M_RESTART : BOOL; (* AT %MW410.1 *)
    GATE11_M_도어_잠김 : BOOL; (* AT %MW410.3 *)
    GATE11_M_비상정지 : BOOL; (* AT %MW410.7 *)
    GATE11_M_이상_리셋 : BOOL; (* AT %MW410.0 *)
    GATE11_M_정상 : BOOL; (* AT %MW410.4 *)
    GATE11_M_정지_CALL : BOOL; (* AT %MW410.2 *)
    GATE11_M_통신_이상 : BOOL; (* AT %MW410.14 *)
    GATE12_M_CP_TRIP : BOOL; (* AT %MW411.15 *)
    GATE12_M_RESTART : BOOL; (* AT %MW411.1 *)
    GATE12_M_도어_잠김 : BOOL; (* AT %MW411.3 *)
    GATE12_M_비상정지 : BOOL; (* AT %MW411.7 *)
    GATE12_M_이상_리셋 : BOOL; (* AT %MW411.0 *)
    GATE12_M_정상 : BOOL; (* AT %MW411.4 *)
    GATE12_M_정지_CALL : BOOL; (* AT %MW411.2 *)
    GATE12_M_통신_이상 : BOOL; (* AT %MW411.14 *)
    GATE_10_M_GATE_OPEN_보조 : BOOL; (* AT %MW409.12 *)
    GATE_11_M_GATE_OPEN_보조 : BOOL; (* AT %MW410.12 *)
    GATE_12_M_GATE_OPEN_보조 : BOOL; (* AT %MW411.12 *)
    GB10_7_10_PLC_BOX_CP_TRIP : BOOL; (* AT %MW87100.15 *) (* 입력 접점 15 *)
    GB10_EPB_비상정지1 : BOOL; (* AT %MW87102.0 *) (* 입력 접점 00 *)
    GB10_EPB_비상정지2 : BOOL; (* AT %MW87102.1 *) (* 입력 접점 01 *)
    GB10_GATE_LOCK_SW_열림1 : BOOL; (* AT %MW87102.8 *) (* 입력 접점 08 *)
    GB10_GATE_LOCK_SW_열림2 : BOOL; (* AT %MW87102.9 *) (* 입력 접점 09 *)
    GB10_PBL_CYCLE_정지 : BOOL; (* AT %MW87100.1 *) (* 입력 접점 01 *)
    GB10_PBL_CYCLE_정지_LP : BOOL; (* AT %MW97101.1 *) (* 출력 접점 01 *)
    GB10_PBL_자동_운전 : BOOL; (* AT %MW87100.0 *) (* 입력 접점 00 *)
    GB10_PBL_자동_운전_LP : BOOL; (* AT %MW97101.0 *) (* 출력 접점 00 *)
    GB10_PB_이상_리셋 : BOOL; (* AT %MW87100.2 *) (* 입력 접점 02 *)
    GB10_SAFETY_DOOR_UNLOOK1 : BOOL; (* AT %MW97103.0 *) (* 출력 접점 00 *)
    GB10_SAFETY_DOOR_UNLOOK2 : BOOL; (* AT %MW97103.1 *) (* 출력 접점 01 *)
    GB10_TL_GREEN_LAMP : BOOL; (* AT %MW97101.9 *) (* 출력 접점 09 *)
    GB10_TL_RED_LAMP : BOOL; (* AT %MW97101.8 *) (* 출력 접점 08 *)
    MCP_M_이상_리셋 : BOOL; (* AT %MW350.4 *)
    MCP_M_자동_START : BOOL; (* AT %MW350.3 *)
    TON_GATE10_OPEN : TON;
    TON_GATE11_OPEN : TON;
    TON_GATE12_OPEN : TON;
    T_GB10_CP_OFF_DELAY : TON;
    T_GB10_통신_이상_DELAY : TON;
    T_GB11_CP_OFF_DELAY : TON;
    T_GB11_통신_이상_DELAY : TON;
    T_GB12_CP_OFF_DELAY : TON;
    T_GB12_통신_이상_DELAY : TON;
    _0006_EB10_CFG_ER : BOOL; (* AT %MW186022.0 *) (* EB 구성 에러 *)
    _0006_EB10_DEER : BOOL; (* AT %MW186022.1 *) (* EB 운전 중 탈락 *)
    _0006_EB10_IO_DEER : BOOL; (* AT %MW186023.2 *) (* EB IO 탈락 에러 *)
    _0006_EB10_IO_TYER : BOOL; (* AT %MW186023.1 *) (* EB IO 타입 에러 *)
    _0007_EB10_CFG_ER : BOOL; (* AT %MW187022.0 *) (* EB 구성 에러 *)
    _0007_EB10_DEER : BOOL; (* AT %MW187022.1 *) (* EB 운전 중 탈락 *)
    _0007_EB10_IO_DEER : BOOL; (* AT %MW187023.2 *) (* EB IO 탈락 에러 *)
    _0007_EB10_IO_TYER : BOOL; (* AT %MW187023.1 *) (* EB IO 타입 에러 *)
    전체_M_GATE_CYCLE_정지 : BOOL; (* AT %MW308.0 *) (* 전체 M GATE CYCLE STOP *)
    전체_M_GATE_비상정지_정상 : BOOL; (* AT %MW308.4 *)
    전체_M_GATE_열림_조건 : BOOL; (* AT %MW308.3 *) (* 전체 M GATE 열림 조건 *)
    전체_M_GATE_자동기동 : BOOL; (* AT %MW308.1 *) (* 전체 M GATE 자동기동 *)
    전체_M_이상_리셋 : BOOL; (* AT %MW308.2 *) (* 전체 M 이상 리셋 *)
    전체_라인_M_총괄_이상 : BOOL; (* AT %MW300.0 *)
END_VAR
VAR
    INST : TON;
END_VAR

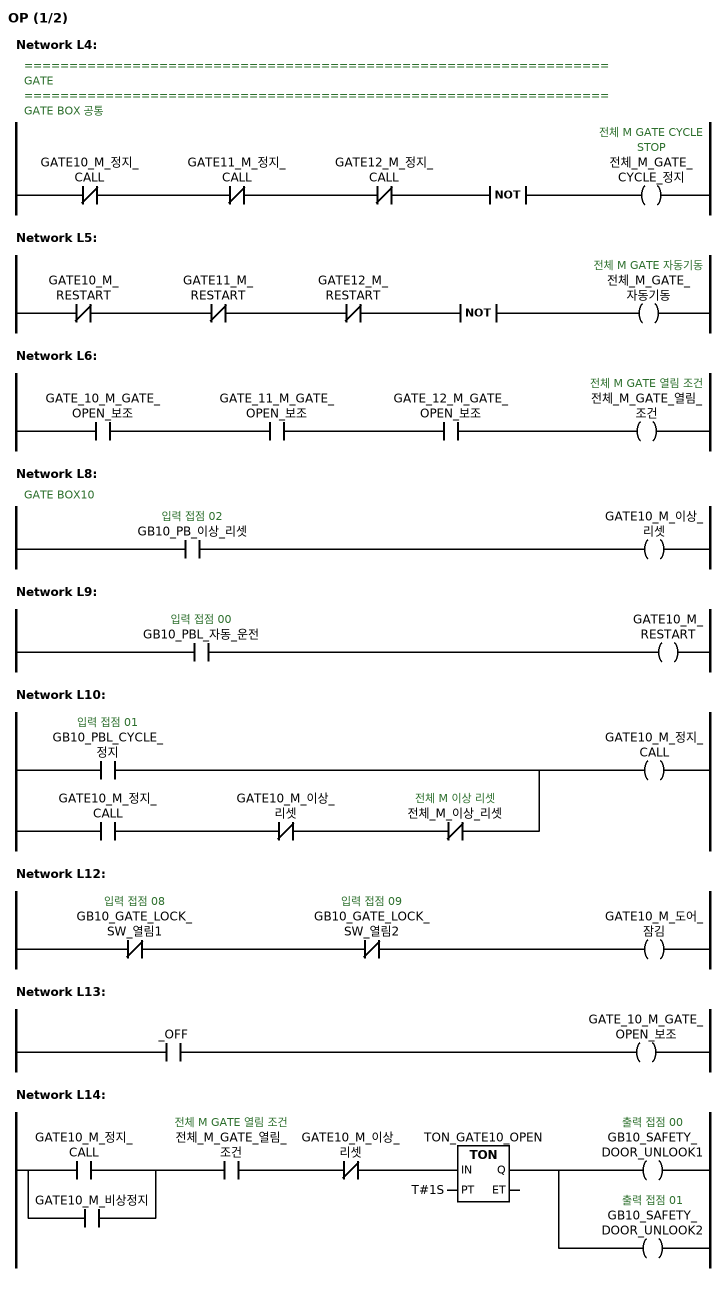
(* ================================================================= *)
(* GATE *)
(* ================================================================= *)
(* GATE BOX 공통 *)
(* Rung L4 *)
전체_M_GATE_CYCLE_정지 := NOT (NOT GATE10_M_정지_CALL AND NOT GATE11_M_정지_CALL AND NOT GATE12_M_정지_CALL);
(* Rung L5 *)
전체_M_GATE_자동기동 := NOT (NOT GATE10_M_RESTART AND NOT GATE11_M_RESTART AND NOT GATE12_M_RESTART);
(* Rung L6 *)
전체_M_GATE_열림_조건 := GATE_10_M_GATE_OPEN_보조 AND GATE_11_M_GATE_OPEN_보조 AND GATE_12_M_GATE_OPEN_보조;
(* GATE BOX10 *)
(* Rung L8 *)
GATE10_M_이상_리셋 := GB10_PB_이상_리셋;
(* Rung L9 *)
GATE10_M_RESTART := GB10_PBL_자동_운전;
(* Rung L10 *)
GATE10_M_정지_CALL := GB10_PBL_CYCLE_정지 OR (GATE10_M_정지_CALL AND NOT GATE10_M_이상_리셋 AND NOT 전체_M_이상_리셋);
(* Rung L12 *)
GATE10_M_도어_잠김 := NOT GB10_GATE_LOCK_SW_열림1 AND NOT GB10_GATE_LOCK_SW_열림2;
(* Rung L13 *)
GATE_10_M_GATE_OPEN_보조 := _OFF;
(* Rung L14 *)
TON_GATE10_OPEN(IN := (GATE10_M_정지_CALL OR GATE10_M_비상정지) AND 전체_M_GATE_열림_조건 AND NOT GATE10_M_이상_리셋, PT := T#1S);
GB10_SAFETY_DOOR_UNLOOK1 := TON_GATE10_OPEN.Q;
GB10_SAFETY_DOOR_UNLOOK2 := TON_GATE10_OPEN.Q;

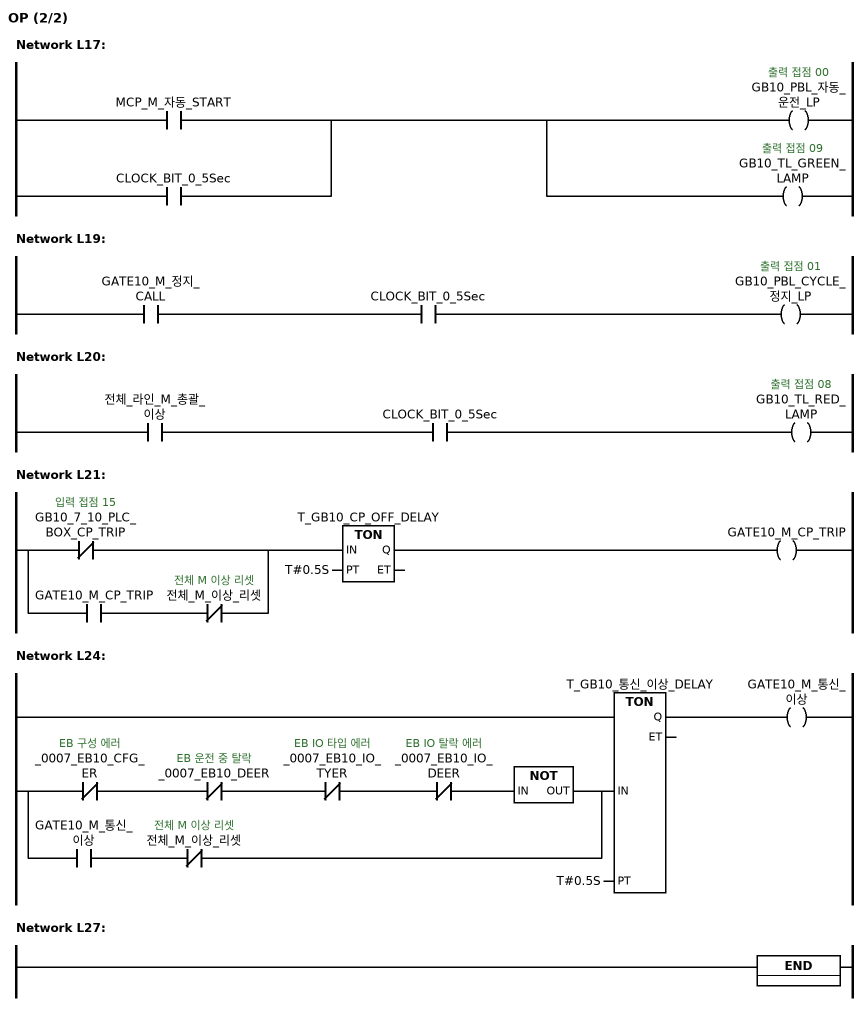
(* Rung L17 *)
GB10_PBL_자동_운전_LP := MCP_M_자동_START OR CLOCK_BIT_0_5Sec;
GB10_TL_GREEN_LAMP := MCP_M_자동_START OR CLOCK_BIT_0_5Sec;
(* Rung L19 *)
GB10_PBL_CYCLE_정지_LP := GATE10_M_정지_CALL AND CLOCK_BIT_0_5Sec;
(* Rung L20 *)
GB10_TL_RED_LAMP := 전체_라인_M_총괄_이상 AND CLOCK_BIT_0_5Sec;
(* Rung L21 *)
T_GB10_CP_OFF_DELAY(IN := NOT GB10_7_10_PLC_BOX_CP_TRIP OR (GATE10_M_CP_TRIP AND NOT 전체_M_이상_리셋), PT := T#0.5S);
GATE10_M_CP_TRIP := T_GB10_CP_OFF_DELAY.Q;
(* Rung L24 *)
T_GB10_통신_이상_DELAY(IN := (NOT (NOT _0007_EB10_CFG_ER AND NOT _0007_EB10_DEER AND NOT _0007_EB10_IO_TYER AND NOT _0007_EB10_IO_DEER)) OR (GATE10_M_통신_이상 AND NOT 전체_M_이상_리셋), PT := T#0.5S);
GATE10_M_통신_이상 := T_GB10_통신_이상_DELAY.Q;
(* Rung L27 *)
END();
END_PROGRAM

PROGRAM 비상정지 (* task: 스캔 프로그램 *)
VAR_EXTERNAL
    AWAYS_ON : BOOL; (* AT %MW3.1 *)
    GATE10_M_도어_잠김 : BOOL; (* AT %MW409.3 *)
    GATE10_M_비상정지 : BOOL; (* AT %MW409.7 *)
    GATE10_M_이상_리셋 : BOOL; (* AT %MW409.0 *)
    GATE10_M_정상 : BOOL; (* AT %MW409.4 *)
    GATE11_M_도어_잠김 : BOOL; (* AT %MW410.3 *)
    GATE11_M_비상정지 : BOOL; (* AT %MW410.7 *)
    GATE11_M_이상_리셋 : BOOL; (* AT %MW410.0 *)
    GATE11_M_정상 : BOOL; (* AT %MW410.4 *)
    GATE12_M_도어_잠김 : BOOL; (* AT %MW411.3 *)
    GATE12_M_비상정지 : BOOL; (* AT %MW411.7 *)
    GATE12_M_이상_리셋 : BOOL; (* AT %MW411.0 *)
    GATE12_M_정상 : BOOL; (* AT %MW411.4 *)
    GB10_EPB_비상정지1 : BOOL; (* AT %MW87102.0 *) (* 입력 접점 00 *)
    GB10_EPB_비상정지2 : BOOL; (* AT %MW87102.1 *) (* 입력 접점 01 *)
    MCP_EPB_비상정지1 : BOOL; (* AT %MW87635.0 *) (* 입력 접점 00 *)
    MCP_EPB_비상정지2 : BOOL; (* AT %MW87635.1 *) (* 입력 접점 01 *)
    MCP_M_비상정지 : BOOL; (* AT %MW350.7 *)
    MCP_M_이상_리셋 : BOOL; (* AT %MW350.4 *)
    R101_1_1_M_I_RB_비상정지 : BOOL; (* AT %MW20040.4 *)
    R101_1_M_I_RB_비상정지 : BOOL; (* AT %MW20070.4 *)
    R101_2_M_I_RB_비상정지 : BOOL; (* AT %MW20060.4 *)
    R101_3_M_I_RB_비상정지 : BOOL; (* AT %MW20050.4 *)
    R102_1_1_M_I_RB_비상정지 : BOOL; (* AT %MW20090.4 *)
    R102_1_M_I_RB_비상정지 : BOOL; (* AT %MW20080.4 *)
    R103_1_M_I_RB_비상정지 : BOOL; (* AT %MW20100.4 *)
    S101_M_총괄_비상정지_이상 : BOOL; (* AT %MW1009.1 *)
    S102_M_총괄_비상정지_이상 : BOOL; (* AT %MW1509.1 *)
    S103_M_총괄_비상정지_이상 : BOOL; (* AT %MW2009.1 *)
    S104_M_총괄_비상정지_이상 : BOOL; (* AT %MW2509.1 *)
    전체_M_GATE_비상정지_정상 : BOOL; (* AT %MW308.4 *)
    전체_M_운전준비_보조 : BOOL; (* AT %MW308.5 *)
    전체_M_이상_리셋 : BOOL; (* AT %MW308.2 *) (* 전체 M 이상 리셋 *)
    전체_OP_M_총괄_비상정지_정상 : BOOL; (* AT %MW304.2 *) (* 전체 OP M 총괄 비상정지 정상 *)
    전체_공정_M_총괄_비상정지_정상 : BOOL; (* AT %MW304.1 *) (* 전체 공정 M 총괄 비상정지 정상 *)
    전체_라인_M_총괄_비상정지_정상 : BOOL; (* AT %MW304.0 *) (* 전체 라인 M 총괄 비상정지 정상 *)
END_VAR

